(* CoDeSys 2.3.9.47 project: PassiProj_V2_3.pro *)
(* Libraries: Ethernet.lib 2.12.10 14:48:32, SerComm.lib 31.5.11 08:54:36, Serial_Interface_01.lib 22.4.13 12:50:14, SysLibEvent.lib 2.12.10 14:48:34, SysLibFile.lib 2.12.10 14:48:34, SysLibPlcCtrl.lib 2.12.10 14:48:32, SysLibSockets.lib 10.2.11 09:20:54, SysLibRtc.lib 2.12.10 14:48:32, Util.lib 26.9.14 11:12:46, Visual.lib 2.12.10 14:48:34, WagoLibStatus.lib 2.12.10 14:48:32, Standard.lib 2.12.10 14:48:34, SYSLIBCALLBACK.LIB 2.12.10 14:48:32 *)

(* PLC configuration (modules and I/O channels)
releLux1 AT %QX2.0 [BOOLOnX_Q] Ch_1 Digital output
releLux2 AT %QX2.1 [BOOLOnX_Q] Ch_2 Digital output
AT %QX2.2 [BOOLOnX_Q] Ch_3 Digital output
AT %QX2.3 [BOOLOnX_Q] Ch_4 Digital output
LUM01 AT %IW0 [WORDOnW_I] Ch_1 Input word
LUM02 AT %IW1 [WORDOnW_I] Ch_2 Input word
LUM03 AT %IW2 [WORDOnW_I] Ch_1 Input word
LUM04 AT %IW3 [WORDOnW_I] Ch_2 Input word
LUM05 AT %IW4 [WORDOnW_I] Ch_1 Input word
LUM06 AT %IW5 [WORDOnW_I] Ch_2 Input word
LUX01 AT %QW0 [WORDOnW_Q] Ch_1 Analog output
LUX02 AT %QW1 [WORDOnW_Q] Ch_2 Analog output
Fieldbus variables [FB_VARS] node 1, in %IB0 out %QB0
Flag variables [FLAG_VARS] node 2, in %IB0 out %QB0
Modbus-Master [MB_MASTER] node 3, in %IB0 out %QB0
*)

(* Global variable list: Global_Constants *)
VAR_GLOBAL CONSTANT

	Plant_NAME			: STRING :='cySN:128 cyVER:1 - ';
	Plant_SN			: DWORD  :=128;	(* S/N Impianto di telecontrollo *)
	Plant_SW_VER		: WORD   :=1;		(* Versione SW installata *)


	(* Colour defines *)
	COLOR_RED			: DWORD	:= 16#2020F0;
	COLOR_YELLOW		: DWORD	:= 16#20F0F0;
	COLOR_GREEN			: DWORD	:= 16#20F020;
	COLOR_LIGHT_GREEN	: DWORD 	:= 16#006000;
	COLOR_GREEN_OFF	 : DWORD	:= 16#108010;

	(* Parameters *)
	Plant_DefaultTAmb	: INT	:=100;		(* [.1°C] Temperatura ambiente di default in caso di rottura sonda *)
	Plant_MaxRunTAmb	: INT   :=210; 		(* [.1°C] Temperatura ambiente massima funzionamento impianto *)
	Plant_AntiFreezeTAmb: INT   :=-40;		(* [.1°C] Antifreeze temperature, start circulators *)
	Plant_VRD_TAlarm	: INT   :=850;(*450;*) 		(* [.1°C] Temperatura di allarme VRD, blocco *)
	Plant_VRD_TMax		: INT   :=800;(*430;*) 		(* [.1°C] Setpoint massimo per uscita VRD *)
	Plant_VRD_TDefault	: INT	:=300;		(* [.1°C] Temperatura di default in caso di errore climatica *)
	Plant_CirOffDelay	: TIME	:=T#30m;	(* (Def.T#15m) Ritardo spegnimento pompe per ricircolo caldaia *)
	Plant_CirOnDelay	: TIME	:=T#15m;
	Plant_MaxWaterLoss	: WORD  :=2;		(* [lt/h] Massima perdita del circuito *)

	(* Filesystem *)
	FilesPath  			: STRING :='S:\';

	(* TCP Logger *)
	Logger_SERVER		: STRING:='';
	Logger_IP				: STRING:= '192.168.100.3';
	Logger_PORT			: WORD  :=80;
	Logger_GETSTART		: STRING:='GET /cygmsrv/passi.ashx?';
	Logger_GETEND		: STRING:='$R$N$R$N';
	Logger_CHECK		: STRING:='True';
	Logger_CRLF			: STRING:='$R$N';
	Logger_DataFile		: STRING:='S:\LOG.DAT';
	Logger_DataFileOld	: STRING:='S:\LOG.BCK';
	Logger_IndexFile	: STRING:='S:\LOG.IDX';
	Logger_ConnRetries	: BYTE:=5;
	Logger_RecoverMsgs	: BYTE:=25;

	(* TCP Remote *)
	Remote_PORT			: WORD  :=10;
	Remote_WELCOME		: STRING:='Connected$R$N';
	Remote_OK			: STRING:='OK$R$N';
	Remote_ERROR		: STRING:='ERROR$R$N';

	(* TCP Sockets *)
	MAX_SEND_TCP_SERVER					 : DWORD:=12000;(*60000*)
	MAX_RECEIVE_TCP_SERVER				 : DWORD:=12000; (*3000;*)
	MAX_RECEIVE_TCP_SERVER_SOCKET	 	 : DWORD:=12000; (* 1500; *)
	MAX_SEND_TCP_CLIENT					 : DWORD:=12000;(*15000*)
	MAX_RECEIVE_TCP_CLIENT				 : DWORD:=12000;
	MAX_RECEIVE_TCP_CLIENT_SOCKET		 : DWORD:=12000;
	MAX_RECEIVE_UDP_SERVER				 : INT  :=1472;
	MAX_RECEIVE_UDP_CLIENT				 : INT  :=1472;
	CONNECT_WATCHDOG_TIME				 : TIME :=t#10s;


	(*  *)
	MAXLUM : BYTE:=2;  (*  6 *)

	(* Lux element *)
	ANALOG		: BOOL:=0;
	DIGITAL			: BOOL:=1;
	MAX_LUXNUM	: WORD := 2;	(* si prevedono al max 100 - 120 lux *)
	LUXM_MAX_ID	: WORD:=250;
	MAX_ARRAY_MSG	: BYTE:=99;

	CRON_MAX	: WORD := 5;



	(* Dim ARRAY retentivi  *)
	MAX_LUX_RETAIN	: BYTE := 250;
	MIN_FOR_DAY: WORD:=1440;
	DOUBLE_MIN_FOR_DAY: WORD:=2880;
	QUARTER_FOR_DAY:WORD:=96;
	DOUBLE_QUARTER_FOR_DAY:WORD:=192;
END_VAR



VAR_GLOBAL
	TestNodoInterogato: BYTE;
	NodoDaInterrogare: BYTE;
	InibiscoModbus: BOOL;
END_VAR

(* Global variable list: Global_Retain *)
VAR_GLOBAL RETAIN PERSISTENT
	Mode_Manual : BOOL := FALSE;
(*
	GRU01_Clima	: typ_Clima;

	VRD01_Clima : typ_Clima;
	VRD02_Clima : typ_Clima;
	VRD03_Clima : typ_Clima;  *)

	Ctl01_Counter	:	DWORD;
	Ctl02_Counter	:	DWORD;
	Ctl03_Counter	:	DWORD;

(* Impostazioni di imipanto *)

	DelayAllarmeTemperaturaNonRaggiunta: INT;
	DeltaInterventoAllarmeTempeaturaNonRaggiuta: INT;
	OffsetSetPointManuale:INT;							(* Offset al Setpoint manuale per comensare lo scambiatore *)

	SogliaMinStartAntigelo: INT;
	SogliaMinStopAntigelo: INT;
	BitAbilitaAntigelo: BOOL:=TRUE;


	GlobalWorkingtime		: ARRAY [1..MAX_LUX_RETAIN] OF DWORD; (* [sec] Internal working time counter *)
	GlobalPowerOnCycles	: ARRAY [1..MAX_LUX_RETAIN] OF WORD;	(*/DWORD;  *) (* Internal counter of power-on cycles *)
	GlobalEnergyCounter	: ARRAY [1..MAX_LUX_RETAIN] OF WORD; (* DWORD;  *) (* [E-1 kWh] Internal energy counter *)
	GlobalEnergyCounter_t 	: ARRAY [1..MAX_LUX_RETAIN] OF DWORD; (* Temporary energy in E-2*Wsec *)

END_VAR

(* Global variable list: Global_Variables *)
VAR_GLOBAL

	SYS    : typ_SYS;
	Logger : typ_Logger;

	T_AMB	:	INT;		(* Environment temperature *)

	Rampa_1, Rampa_2	: RAMP_INT;
	RampUp			:INT:=500;
	RampDown			:INT:=500;
	RampTime			:TIME:= t#500ms;



	(**** PLANT OBJECTS ****)
	(*...*)
(*	GRU01	:	obj_CAL_VT300GW2 := (ID:=1); *)

	(* Water counter - 2 PULSES/LITER *)

	(* Heat counter *)

	(* Cronothermostat *)
(*	THER01	:	obj_CRONTER := (ID:=1, Local_MaxRunTAmb:=250,Histeresys:=10);
	THER02	:	obj_CRONTER := (ID:=2, Local_MaxRunTAmb:=250,Histeresys:=10);
	THER03	:	obj_CRONTER := (ID:=3, Local_MaxRunTAmb:=250,Histeresys:=10);
	THER04	:	obj_CRONTER := (ID:=4, Local_MaxRunTAmb:=600,Histeresys:=10);	(* There is no an environment probe	*)
	THER05	:	obj_CRONTER := (ID:=5, Local_MaxRunTAmb:=800,Histeresys:=50);	(*  crono per la gestione della caldaia a muro ex CAL04 ora CIR250 *)
	THER250	:	obj_CRONTER := (ID:=250, Local_MaxRunTAmb:=800,Histeresys:=50);	(*  crono per la gestione della caldaia a muro ex CAL04 ora CIR250 *)


	 Boiler *)

	(* Pump *)

	(* Modbus double pumps *)

	(* ModBus Pumps *)

	(* Valves
	VRD01	:	obj_VRD_new 	:= (ID:=1, fFeedback:=TRUE, ReducedRange := TRUE,Local_VRD_TAlarm:=450);
	VRD02	:	obj_VRD_new 	:= (ID:=2, fFeedback:=TRUE, ReducedRange := TRUE,Local_VRD_TAlarm:=450);
	VRD03	:	obj_VRD_new 	:= (ID:=3, fFeedback:=TRUE, ReducedRange := TRUE,Local_VRD_TAlarm:=850);
 *)

	TolleranceLowLux	:WORD :=2; (* Tolleranza per isteresi in Lux - era 25 *)
	TolleranceHighLux	:WORD :=2; (* Tolleranza per isteresi in Lux  - era 25 *)

	(* Lux probes *)
	LumList : ARRAY [1..6] OF obj_LUM;

	LuxElement		: ARRAY [1..MAX_LUXNUM] OF obj_LUX;  (* Lista di variabili Lux   *)

	DataLuxForVis	: ARRAY [1..MAX_LUXNUM] OF type_DataLuxForVis;	(*ARRAY ordinato contenente i valori Status_Vis e del timer utilizzati per la visualizzazione (PLC_Visualization)*)

	LuxOutput		: ARRAY [1..LUXM_MAX_ID] OF type_LuxOutput;

	(* Crono *)
	CRON   			: ARRAY [1..CRON_MAX] OF obj_CRON;
	CronEd			: obj_CRON_EDITOR;
	LuxSuBit		: REAL:= 0.15259;  (* 60000 / 32767= 1.83111 *) (* 5000 / 32767= 0.15259 *)  (* 1000 / 32767= 0.03 *)

	(** Communication **)
	(**** SIMULATION ONLY ****)
	(*...*)END_VAR

(* Data type in Lux *)
TYPE en_ActionKey :
(
	NormalMode 	:= 0,
	SwitchON		:= 1,
	SwitchOFF		:= 2,
	Restore			:= 3
);
END_TYPE

(* Data type in Lux *)
TYPE en_KeyMode :
(
	BUTTON_NO		:=01,
	BUTTON_NC		:=02,
	SWITCH_NO		:=03,
	SWITCH_NC			:=04
);
END_TYPE

(* Data type in Logger *)
TYPE en_Logger_ErrLev :
(
	EL_Log			:=0,
	EL_Wrn			:=1,
	EL_Alarm		:=2,
	EL_AlarmStop	:=3
);
END_TYPE

(* Data type in Logger *)
TYPE en_Logger_Status :
(
	S_Logger_UNKNOWN := 0,
	S_Logger_IDLE,
	S_Logger_WAITCONN,
	S_Logger_WAITTX,
	S_Logger_WAITRESP,
	S_Logger_ERROR
);
END_TYPE

(* Data type in Lux *)
TYPE en_Modality :
(
	ManualeOff 	:= 0,
	ManualeOn 	:= 1,
	Cronografo	:= 2,
	Timer		:= 3,
	KeyControl	:= 4
);
END_TYPE

(* Data type *)
TYPE en_SYS_Objects :
(
	EO_SYS		:=0,  (* PLC *)
	EO_VPN		:=1,  (* VPN *)
	EO_DOOR		:=2,  (* Door & access control *)

	EO_CAL		:=10, (* Caldaia *)
	EO_CIR		:=11, (* Circolatore *)
	EO_CRON		:=12, (* Crono-termostato *)
	EO_VRD		:=13, (* Valvola miscelatore pannelli *)
	EO_CTL		:=14, (* Contalitri *)
	EO_CTB		:=15, (* Contabilizzatore *)
	 (*EO_TPV		:=16, Temperature probes values *)
	EO_PPV		:=17, (* Pressure probes values *)
	EO_PBV		:=18, (* Over-Pressure Alarms *)
	EO_TBV		:=19, (* Over-Temperature Alarms *)
	EO_PMV		:=20, (* Under-Pressure Alarms *)
	EO_GRU		:=21, (* Gruppo termico *)
	EO_PDC		:=22, (* Pompa di calore *)
	EO_SOL		:=23, (* Pannello solare termico *)
	EO_ESOL		:=24, (* Pannello solare fotovoltaico *)
	EO_GAS		:=25, (* Contatore GAS *)
	EO_PORT		:=26, (* Misuratore di portata *)
	EO_FPV		:=27, (* Flow probes values *)
	EO_ANZ		:=28, (* Analizzatore di rete *)
	EO_SCA		:=29, (* Signal Control Alarms *)
	EO_LUX		:=30, (* Base Illumination point *)
	EO_LUXM		:=31, (* Metered Illumination point *)
	EO_PSG		:=32, (* Sensore di passaggio *)
	EO_HVAC		:=33, (* Heating, Ventilating and Air Conditioning *)
	EO_HYGRV	:=34, (* Relative Humidity sensors value *)
	EO_COOV		:=35, (* Carbon Dioxide CO2 sensors value *)
	EO_INV		:=36, (* Inverter *)
	EO_STR		:=37, (* Smart string box *)

	EO_CIRD		:=39, (* Double CIR *)
	EO_ACS		:=40, (* Hot domestic water *)
	EO_FRG		:=41, (* Frigo *)
	EO_THER		:=42, (* Thermostat *)
	EO_CIRM		:=43, (* Modbus CIR *)

	EO_LUM		:=16, (* Lumen *)

	EO_ZGW			:=200,  (* ZigBee - Gateway *)
	EO_ZRM			:=201,	(* ZigBee - Repeater *)
	EO_ZREL			:=202,	(* ZigBee - Actuator rele *)
	EO_ZTHL			:=203,	(* ZigBee - Temperature Sensor *)

	EO_ASGW			:=250,	(* ASi - Gateway *)
	EO_ASCBI		:=251,	(* ASi - Input Board, Ciabatta *)

	EO_LON			:=1000, (* Bus - LON *)
	EO_MODBUS		:=1001, (* Bus - MODBUS *)
	EO_MBUS			:=1002, (* Bus - M-BUS *)
	EO_MODBUS_TCP	:=1003, (* Bus - MODBUS TCP *)

	EO_GENERIC		:=9000, (* Generic dataset *)
	EO_EXPO			:=9001 (* EXPO dataset *)
);
END_TYPE

(* Data type *)
TYPE en_SYS_Status :
(
	S_UNKNOWN  := 0,
	S_STARTUP,
	S_INIT_RTC,
	S_INIT_VAR,
	S_AUTOTEST,
	S_RUNNING,
	S_SHUTDOWN,
	S_HALT
);
END_TYPE

(* Data type in Plant_Objects *)
TYPE typ_Cron_Calendar :
STRUCT
	Profile		: ARRAY[0..384] OF BYTE;
END_STRUCT
END_TYPE

(* Data type in Plant_Objects *)
TYPE typ_Cron_Jolly :
STRUCT
	Start		: DT;
	End			: DT;
	Temp		: WORD;
	Flags		: WORD; (* B0:Enabled B1..B15:Unused *)
END_STRUCT
END_TYPE

(* Data type in Plant_Objects *)
TYPE typ_Cron_Profile :
STRUCT
	Flags		: WORD;
	Setpoint	: ARRAY [0..1439] OF WORD;	(*	Setpoint	: ARRAY [0..95] OF WORD;  *)
END_STRUCT
END_TYPE

(* Data type in Logger *)
TYPE typ_Logger :
STRUCT
	Status		: en_Logger_Status;

	SendReq		: BOOL;
	SendIdx		: DWORD;
	SendData	: ARRAY [0..MAX_SEND_TCP_CLIENT] OF BYTE;
	SendLen		: DINT;

	TData		: ARRAY [0..MAX_SEND_TCP_CLIENT] OF BYTE;
	TLen		: DINT;

	LastIdxPos	: DWORD;

	(* Temporary variables used by objects *)
	s1			: STRING(256);
	i1			: WORD;

END_STRUCT
END_TYPE

(* Data type *)
TYPE typ_SYS :
STRUCT
	Status			: en_SYS_Status;
	Warning			: BOOL;
	Alarm			: BOOL;
	AlarmStop		: BOOL;

	Time_LogString	: STRING;
	Time_Year		: WORD;
	Time_Month		: BYTE;
	Time_Day		: BYTE;
	Time_Hour		: BYTE;
	Time_Minute		: BYTE;
	Time_Min		: BYTE;

	Time_CT_DT		: DT;
	Time_CT_Day		: WORD;
	Time_CT_Quarter	: BYTE;
	Time_CT_Minute		: WORD;

	LastLogs_Idx	: BYTE;
	LastLogs_Dat	: ARRAY[0..5] OF STRING;
	LastLogs_Msg	: ARRAY[0..5] OF STRING;

END_STRUCT
END_TYPE

(* Data type in Lux *)
(* La seguente struttura ha la funzione di collegare l'id del lux con i relativi dati qui indicati *)
(* In tal modo la visualizzazione dello stato dei lux viene eseguita associando l'ID dell'array contenente questa struttura*)

TYPE type_DataLuxForVis :
STRUCT
	VisStatus	: DWORD; (* valori di status_vis   *)
	VisTimer	: TIME;	(* Valori dei timer  *)
	VisMod		: en_Modality; (* Impostazione mode  *)
END_STRUCT
END_TYPE

(* Data type in Lux *)
TYPE type_LuxOutput :
STRUCT
	DigitalOut	:	BOOL;
	AnalogOut	:	WORD;
	TypeOut	:	BOOL;
END_STRUCT
END_TYPE

(* POU PLC_PRG, ST *)
PROGRAM PLC_PRG
VAR
	Timer1: TON; (* Fast controls tick *)
	Timer2: TON; (* Plant control tick *)
	Timer3: TON; (* Logger timer *)
	Timer4: TON; (* Media timer *)

	LumValue			: ARRAY [1..6] OF WORD;
	LumValueSum		: DWORD;
	LumValueMax, LumValueMin	: WORD;
	LumValueAverage	: DWORD;
	LumValueAverageLux	:DWORD;
	LuxDeltaBit, LuxEndBit	:WORD;
	x					: BYTE;
	counter				: WORD;
	LuxCount			: WORD;
	LuxEnInfo	: BOOL;
	ValInCrono	: INT; (* Valore del setpoint del crono *)

	TolleranceLowBit		: WORD;
	TolleranceHighBit		: WORD;
	AnalogOutputBit			:WORD;

	ValInCronoVisu			:ARRAY [1..MAX_LUXNUM] OF INT;
	ValInCronoFromVisu		:ARRAY  [1..MAX_LUXNUM] OF BOOL;
	Temp	:INT;
	LuxStateON: BOOL;
END_VAR
(******************************************************************************
 ****                           MAIN TASK CODE                             ****
 ******************************************************************************

	Network setup:
		IP  = 192.168.100.2 | MSK = 255.255.255.0
		GW	= 192.168.100.1 | DNS = 192.168.100.1
		SNTP = 193.204.114.232 (3600s) ==> 192.168.100.3

*)

(*==============================*)
(*===== Main status machine ====*)
(*==============================*)
MainCtrl();
(*
IF SYS.Status>S_INIT_VAR THEN
	Execute cycle processes
END_IF
 *)
(*==============================*)
(*== System cycle operations ===*)
(*==============================*)
(* Execute TCP processes *)
Logger_Proc();
Remote_Proc();
(* Execute Cron Editor commands *)
CronEd();
END_PROGRAM
ACTION MainCtrl:
CASE Sys.Status OF

	S_STARTUP:
		Sys.Status:=S_INIT_RTC;
		FOR counter := 1 TO MAX_LUXNUM DO
			CRON[counter].ID:=counter;
			LuxElement[counter].ID:=counter;
			LuxElement[counter].CTRL_MODE := 2 ; (* TabDefaultLux[counter].Mode; //copio il mode nella tabella delle variabili dei lux 	*)
			LuxElement[counter].CTRL_MODE_backUp := 2;  (* TabDefaultLux[counter].Mode; //salvo il mode di backup per il ripristina modo	*)
			LuxElement[counter].DimmingType:=1; (* settato a dimming *)
		END_FOR
		FOR x:= 1 TO MAXLUM DO
			LumList[x].ID:= x;
		END_FOR
	S_INIT_RTC:
		(* Check RTC and update from network *)
		RTC_Update();
		(* Check time *)
		IF Sys.Time_Year>2000 THEN
			Sys.Status:=S_INIT_VAR;
		END_IF

	S_INIT_VAR:
		LogEv(EL_Wrn,EO_SYS,0,1,CONCAT('System_startup_v',WORD_TO_STRING(Plant_SW_VER)));
		Sys.Status:=S_RUNNING;

	S_RUNNING:
		Timer1(IN:=NOT Timer1.Q,PT:=T#50ms);
		IF Timer1.Q THEN
			(* Update meters *)

			(* Update system checks *)
			SYS_Proc();
		END_IF

		Timer2(IN:=NOT Timer2.Q,PT:=T#500ms);
		IF Timer2.Q THEN
			(* Read current date/time *)
			RTC_Update();


			(*Lum Probes *)
			IF ValInCronoFromVisu[1] = TRUE THEN
				LumList[1](IN:=LUM01, IN_TARGET:=ValInCronoVisu[1]*10);
			ELSE
				CRON[1]( SetPoint=>ValInCrono);
				LumList[1](IN:=LUM01, IN_TARGET:=ValInCrono);
			END_IF
			IF ValInCronoFromVisu[2] = TRUE THEN
				LumList[2](IN:=LUM02, IN_TARGET:=ValInCronoVisu[2]*10);
			ELSE
				CRON[2]( SetPoint=>ValInCrono);
				LumList[2](IN:=LUM02, IN_TARGET:=ValInCrono);
			END_IF
			LumValue[1]:=LumList[1].AVG;
			LumValue[2]:=LumList[2].AVG;
		(*	LumList[3](IN:=LUM03);
			LumValue[3]:=LumList[3].AVG;
			LumList[4](IN:=LUM04);
			LumValue[4]:=LumList[4].AVG;
			LumList[5](IN:=LUM05);
			LumValue[5]:=LumList[5].AVG;
			LumList[6](IN:=LUM06);
			LumValue[6]:=LumList[6].AVG;
		 *)
			Timer4(IN:=NOT Timer4.Q,PT:=T#500ms);
			IF Timer4.Q THEN
				LumValueSum:=0;
				FOR x:= 1 TO MAXLUM DO
					LumValueSum:= LumValueSum+ LumValue[x];
				END_FOR
				LumValueAverage:=(LumValueSum / MAXLUM);
				LumValueAverageLux:=REAL_TO_DWORD(LumValueAverage*LuxSuBit);
			END_IF

			TolleranceLowBit := REAL_TO_WORD (TolleranceLowLux / LuxSuBit);
			TolleranceHighBit := REAL_TO_WORD (TolleranceHighLux / LuxSuBit);

		FOR LuxCount:=1 TO  MAX_LUXNUM DO
			IF  LuxElement[LuxCount].ID <> 0  THEN (* esegue scansione dei lux dell'impianto solo se presenti *)
	
				CASE LuxElement[LuxCount].CTRL_MODE OF
					0: (* Manuale Off *)
					LuxElement[LuxCount](LuxTypeOut => LuxOutput[LuxCount].TypeOut,
											LuxDigitalOut => LuxOutput[LuxCount].DigitalOut,
											LuxAnalogOut => LuxOutput[LuxCount].AnalogOut,
											Lux_Enable=>LuxEnInfo,
											LocalWorkingTime:=GlobalWorkingtime[LuxCount],
											LocalPowerOnCycles:=GlobalPowerOnCycles[LuxCount],
											LocalEnergyCounter:=GlobalEnergyCounter[LuxCount],
											LocalEnergyCounter_t:=GlobalEnergyCounter_t[LuxCount],KeyQty:=2);
					1:  (* Manuale On *)
					LuxElement[LuxCount](LuxTypeOut => LuxOutput[LuxCount].TypeOut,
											LuxDigitalOut => LuxOutput[LuxCount].DigitalOut,
											LuxAnalogOut => LuxOutput[LuxCount].AnalogOut,
											Lux_Enable=>LuxEnInfo,
											LocalWorkingTime:=GlobalWorkingtime[LuxCount],
											LocalPowerOnCycles:=GlobalPowerOnCycles[LuxCount],
											LocalEnergyCounter:=GlobalEnergyCounter[LuxCount],
											LocalEnergyCounter_t:=GlobalEnergyCounter_t[LuxCount],KeyQty:=2);
					2:	(* se il mode è settato come cronografo gestisco accensione a orologio *)
					CRON[LuxCount]( SetPoint=>ValInCrono);
					(*	LuxElement[LuxCount].ValInCronoInLux:=ValInCrono;   *)
					IF ValInCronoFromVisu[LuxCount] = TRUE THEN
						LuxElement[LuxCount].ValInCronoInLux:=ValInCronoVisu[LuxCount]*10;
					ELSE
						LuxElement[LuxCount].ValInCronoInLux:=ValInCrono;
					END_IF
			(*		KeyTest((*KeyMode:= 01,*)CtrlKey:=LUX_ST[108],Cmd_Enable=>LuxEnInfo );
					KeyTest1((*KeyMode:= 01,*)CtrlKey:=LUX_ST[107],Cmd_Enable=>LuxEnInfo1 );				
					LuxElement[LuxCount].CtrlKeyList[0]:=LuxEnInfo;
					LuxElement[LuxCount].CtrlKeyList[1]:=LuxEnInfo1;								 *)
					LuxElement[LuxCount](LuxTypeOut => LuxOutput[LuxCount].TypeOut,
											LuxDigitalOut => LuxOutput[LuxCount].DigitalOut,
											LuxAnalogOut => LuxOutput[LuxCount].AnalogOut,
											Lux_Enable=>LuxEnInfo,
											LocalWorkingTime:=GlobalWorkingtime[LuxCount],
											LocalPowerOnCycles:=GlobalPowerOnCycles[LuxCount],
											LocalEnergyCounter:=GlobalEnergyCounter[LuxCount],
											LocalEnergyCounter_t:=GlobalEnergyCounter_t[LuxCount],KeyQty:=2);  (*, KeyMode:=KeyTest.KeyMode); *)
				END_CASE
				AnalogOutputBit:= REAL_TO_WORD( LuxOutput[LuxCount].AnalogOut*3.27);
				(* codice non in uso - start *)
				IF  AnalogOutputBit < 3100  THEN
					LuxStateON:=FALSE;	(* se devo aprire il relè per spegnere *)
				ELSIF  AnalogOutputBit  > 3600 THEN
					LuxStateON:=TRUE;	(* se devo chiudere il relè per accendere *)
				END_IF
				(* codice non in uso - end *)
				IF ( AnalogOutputBit > TolleranceLowBit) AND  (AnalogOutputBit < (32767-TolleranceHighBit) ) THEN
					IF  ( LuxOutput[LuxCount].AnalogOut>0 AND
						( ( LumValueAverage<AnalogOutputBit - TolleranceLowBit) OR ( LumValueAverage>AnalogOutputBit + TolleranceHighBit) ))THEN
							IF ( LumValueAverage>AnalogOutputBit + TolleranceHighBit) THEN  (* se il valore medio misurato è maggiore del target impostato  *)
								LuxDeltaBit:=  DWORD_TO_WORD(LumValueAverage)-AnalogOutputBit; (* calcolo diff tra misura e target  *)
								IF LuxDeltaBit < AnalogOutputBit THEN  (* se il delta è minore del target posso sottrarla al target altrimenti azzero l'uscita (posta a 1 bit)  *)
									LuxEndBit:= AnalogOutputBit - LuxDeltaBit;
										(*LuxStateON:=TRUE; se devo chiudere il relè per accendere *)
								ELSE
									 LuxEndBit := 1;
									 (* LuxStateON:=FALSE;	se devo aprire il relè per spegnere *)
								END_IF
								(* LuxEndBit:=REAL_TO_INT(LuxOutput[LuxCount].AnalogOut*3.27) - LuxDeltaBit;  *)
							ELSIF ( LumValueAverage<AnalogOutputBit - TolleranceHighBit) THEN
								LuxDeltaBit:= DWORD_TO_WORD( AnalogOutputBit - LumValueAverage);
								LuxEndBit:= AnalogOutputBit + LuxDeltaBit;
								(* LuxStateON:=TRUE;	 se devo chiudere il relè per accendere *)
								(* LuxEndBit:=REAL_TO_INT(LuxOutput[LuxCount].AnalogOut*3.27) + LuxDeltaBit;  *)
							END_IF;
							CASE LuxCount OF
								1:	IF luxEndBit >32727 THEN
										LuxEndBit:=32727;
									END_IF
									 (*releLux1:=LuxStateON;   apro il contatto del relè se il lux è spento *)
								 	Rampa_1(in:= LuxEndBit, ascend:=RampUp, descend:=RampDown, timebase:=RampTime);
								(*Rampa_1(in:= REAL_TO_INT(LuxOutput[LuxCount].AnalogOut*3.27), ascend:=RampUp, descend:=RampDown, timebase:=RampTime);*)
									 LUX01:=Rampa_1.OUT;

								(*		1: LUX01:= REAL_TO_WORD(LuxOutput[LuxCount].AnalogOut*3.27);	*)
								2:  IF luxEndBit >32727 THEN
										LuxEndBit:=32727;
									END_IF
									 (*releLux1:=LuxStateON;   apro il contatto del relè se il lux è spento *)
									Rampa_2(in:= LuxEndBit, ascend:=RampUp, descend:=RampDown, timebase:=RampTime);
								(*Rampa_2(in:= REAL_TO_INT(LuxOutput[LuxCount].AnalogOut*3.27), ascend:=RampUp, descend:=RampDown, timebase:=RampTime);*)
									 LUX02:=Rampa_2.OUT;
								(*		 LUX02:= REAL_TO_WORD(LuxOutput[LuxCount].AnalogOut*3.27);	*)
							END_CASE;

					END_IF
				ELSIF ( (AnalogOutputBit > (32767-TolleranceHighBit) ) OR ( AnalogOutputBit < TolleranceLowBit) ) THEN
						CASE LuxCount OF
							1: Rampa_1(in:= REAL_TO_INT(LuxOutput[LuxCount].AnalogOut*3.27), ascend:=RampUp, descend:=RampDown, timebase:=RampTime);
								 LUX01:=Rampa_1.OUT;
							2: Rampa_2(in:= REAL_TO_INT(LuxOutput[LuxCount].AnalogOut*3.27), ascend:=RampUp, descend:=RampDown, timebase:=RampTime);
								 LUX02:=Rampa_2.OUT;
						END_CASE;
				END_IF
(*
				IF Rampa_1.OUT  < 3000  OR Rampa_2.OUT < 3000 THEN (* 3100 *)
					releLux1:=FALSE;
				ELSIF( Rampa_1.OUT >3200 OR Rampa_2.OUT > 3200) THEN  (*  3600 *)
					 releLux1:=TRUE;
				END_IF
 *)
				IF (Rampa_1.OUT  < 3000)  THEN (* 3100 *)
					releLux1:=FALSE;
				ELSIF( Rampa_1.OUT >3200 ) THEN  (*  3600 *)
					 releLux1:=TRUE;
				END_IF
				IF (Rampa_2.OUT  < 3000)  THEN (* 3100 *)
					releLux2:=FALSE;
				ELSIF( Rampa_2.OUT >3200 ) THEN  (*  3600 *)
					 releLux2:=TRUE;
				END_IF

			END_IF
		END_FOR



			(* Test toggle *)
			(*IF TEST1 THEN TEST1:=FALSE; ELSE TEST1:=TRUE; END_IF*)
		END_IF

		Timer3(IN:=NOT Timer3.Q,PT:=T#1m);
		IF Timer3.Q THEN
			(* Trig logger *)
			LogTrig();
			(* Execute temporary CSV logger *)
			(*CSV_Log();*)
		END_IF

	S_SHUTDOWN:
		(* Stop sistema *)
		Sys.Status:=S_STARTUP;

	S_HALT:
		(* Aspetta uscita manuale *)
		Sys.Status:=S_STARTUP;

	S_UNKNOWN:
	Sys.Status:=S_STARTUP;
ELSE
	Sys.Status:=S_STARTUP;
END_CASE;
END_ACTION

(* POU TCP_Logger/Logger_Proc, ST *)
PROGRAM Logger_Proc
VAR
	c1:         	TCPCLIENT;

	Open:	    	BOOL;
	IpAddr:			DWORD;
	InetAddr:		DWORD;
	Connected:  	BOOL;
	Error:      	DINT;
	TxTrig:     	BOOL;
	RxData:			ARRAY [0..MAX_RECEIVE_TCP_CLIENT] OF BYTE;
	RxLen:			DINT;

	Retry:			BYTE;	(* Counter for connection retries *)
	Recovered:		BYTE;	(* Counter for recovered unsent messages *)

	i:				DINT;
	pos:			DWORD;
	hFile:			DWORD;

END_VAR
(*=== State machine ===*)
CASE Logger.Status OF

	S_Logger_UNKNOWN:
		(* Startup *)
		Logger.SendReq:=FALSE;
		Open:=FALSE;
		Logger.Status:=S_Logger_IDLE;

	S_Logger_IDLE:
		(* Wait request *)
		IF Logger.SendReq THEN
			(* Resolve server name or use static IP *)
			IF LEN(Logger_SERVER)=0 THEN
				InetAddr:=SysSockInetAddr(Logger_IP);
			ELSE
				IpAddr:=SysSockGetHostByName(ADR(Logger_SERVER));
				DWORDSWAP(pIn:=ADR(IpAddr), pOut:=ADR(InetAddr));
			END_IF
			TxTrig:=FALSE;
			RxLen:=0;
			(* Open connection *)
			Open:=TRUE;
			Logger.Status:=S_Logger_WAITCONN;
		END_IF

	S_Logger_WAITCONN:
		(* Wait connection *)
		IF Connected THEN
			(* Send data *)
			TxTrig:=TRUE;
			Logger.Status:=S_Logger_WAITTX;
		END_IF
		IF Error>0 THEN
			Open:=FALSE;
			Logger.Status:=S_Logger_ERROR;
		END_IF

	S_Logger_WAITTX:
		(* Wait transmission *)
		IF NOT TxTrig THEN
			Logger.Status:=S_Logger_WAITRESP;
		END_IF
		IF Error>0 THEN
			Open:=FALSE;
			Logger.Status:=S_Logger_ERROR;
		END_IF

	S_Logger_WAITRESP:
		(* Wait response *)
		IF Connected=FALSE (* OR TIMEOUT!! *) THEN
			Open:=FALSE;
			(* Check response *)
			IF RxLen>=4 AND CHKSTRING(pString:=ADR(RxData), pPattern:=ADR(Logger_CHECK)) THEN
				Logger.SendReq:=FALSE;
				Retry:=0;
				(* Check unsent messages to flush *)
				IF Recovered<Logger_RecoverMsgs THEN
					MsgChk();
					IF Logger.SendReq=TRUE THEN
						Recovered:=Recovered+1;
					ELSE
						Recovered:=0;
					END_IF
				ELSE
					Recovered:=0;
				END_IF
				Logger.Status:=S_Logger_IDLE;
			ELSE
				Logger.Status:=S_Logger_ERROR;
			END_IF
		END_IF

	S_Logger_ERROR:
		(* Connection error or send failure *)
		Retry:=Retry+1;
		IF Retry>Logger_ConnRetries THEN
			(* Save message as unsent *)
			MsgSave();
			Logger.SendReq:=FALSE;
			Retry:=0;
		END_IF
		Logger.Status:=S_Logger_IDLE;

ELSE
	Logger.Status:=S_Logger_UNKNOWN;
END_CASE


(*=== Execute client lib ===*)
c1(
	xOpenConnection			:= Open,
	dwInetAddr 				:= InetAddr,
	wPortNumber				:= Logger_PORT,
	ptSendData				:= ADR(Logger.SendData),
	diSendCount				:= Logger.SendLen,
	tConnectWatchdogTime	:= t#10s,
	xStartSend				:= TxTrig,
	aReceiveBuffer			:= RxData,
	diReceiveCount			:= RxLen,
	xConnected				=> Connected,
	diError					=> Error
);

(*=== Process Rx data ===*)
(*IF RxLen>0 THEN
	RxLen:=0;
END_IF*)
END_PROGRAM
ACTION MsgChk:
(* Open index file *)
hFile:=SysFileOpen(Logger_IndexFile,'r');
IF hFile=0 THEN
	RETURN;
END_IF
(* Search oldest message to recover *)
SysFileSetPos(hFile,Logger.LastIdxPos);
Logger.SendLen:=0;
REPEAT
	SysFileRead(hFile, ADR(Logger.SendIdx), SIZEOF(Logger.SendIdx));
	pos:=SysFileGetPos(hFile);
	SysFileRead(hFile, ADR(Logger.SendLen), SIZEOF(Logger.SendLen));
UNTIL
	SysFileEOF(hFile) OR Logger.SendLen<>0
END_REPEAT
SysFileClose(hFile);
(* Delete index file when all messages are recovered *)
IF Logger.SendLen=0 THEN
	Logger.LastIdxPos:=0;
	SysFileDelete(Logger_IndexFile);
	RETURN;
END_IF
(* Recover message data *)
hFile:=SysFileOpen(Logger_DataFile,'r');
IF hFile<>0 THEN
	SysFileSetPos(hFile,Logger.SendIdx);
	SysFileRead(hFile,ADR(Logger.SendData),Logger.SendLen);
	Logger.SendReq:=TRUE;
	SysFileClose(hFile);
END_IF
(* Clear index entry *)
hFile:=SysFileOpen(Logger_IndexFile,'a');
IF hFile<>0 THEN
	SysFileSetPos(hFile,pos);
	i:=0;
	SysFileWrite(hFile, ADR(i), 4);
	Logger.LastIdxPos:=SysFileGetPos(hFile);
	SysFileClose(hFile);
END_IF
END_ACTION
ACTION MsgSave:
(* Add log position in recovery indexes *)
hFile:=SysFileOpen(Logger_IndexFile,'a');
SysFileWrite(hFile, ADR(Logger.SendIdx), SIZEOF(Logger.SendIdx));
SysFileWrite(hFile, ADR(Logger.SendLen), SIZEOF(Logger.SendLen));
SysFileClose(hFile);
END_ACTION

(* POU Utils Functions/TCPCLIENT, ST *)
FUNCTION_BLOCK TCPCLIENT
(***********************************************************************************************************	*)
(* Version: 1.3b                        			          													*)
(* Date: 28.10.2014                   				          							            			*)
(***********************************************************************************************************	*)
(* WAGO Kontakttechnik GmbH Hansastr. 27 32423 Minden(Westf.)													*)
(* Tel. +0049 571/887-0 Fax. +0049 571/887-0																	*)
(* Author: VB																									*)
(***********************************************************************************************************	*)
(*Description:	A TCP client to read and write data with additional connection watchdog							*)
(*History:																										*)
(*Version 1.3b: 28.10.2014: Use DWORD address for IP (Andrea Ravasio)											*)
(*Version 1.3: 11.02.2011: Changes according to 750-880/881											 			*)
(*Version 1.2: 29.08.2007 Bugfix TCP Client																		*)
(*Version 1.1: 15.01.2007 Changes according to FW11																*)
(*Version 1.0: 09.03.2006 Release																				*)
(***********************************************************************************************************	*)
VAR CONSTANT
	STATE_CREATE     				 : BYTE:= 0;
	STATE_OPEN     					 : BYTE:= 1;
	STATE_IOCTL    					 : BYTE:= 2;
	STATE_CONNECT     				 : BYTE:= 10;
	STATE_TX       					 : BYTE:= 20;
	STATE_RX       					 : BYTE:= 30;
	STATE_CLOSE    					 : BYTE:= 40;
	STATE_ERROR_TRAP			     : BYTE:= 200;
END_VAR

VAR_INPUT
	xOpenConnection					: BOOL;
	dwInetAddr						: DWORD; (* <== Use SysSockInetAddr() value or
													swapped bytes order of SysSockGetHostByName() value *)
	wPortNumber						: WORD;
	ptSendData						: POINTER TO ARRAY[0..MAX_SEND_TCP_CLIENT] OF BYTE;
	diSendCount						: DINT;
	tConnectWatchdogTime		    : TIME := t#10s;
END_VAR
VAR_OUTPUT
	xConnected						: BOOL;
	diError 						: DINT := 0;
END_VAR
(* ErrorCodes -----------------------------------------
	16#8001 => No socket descriptor available 
	16#8002 => SysSockSend returns -1 
	16#8003 => Socket was "gracefully closed" 
	16#8004 => switching to none blocking mode fails
	16#8005 => SysSockClose() returns FALSE 
    16#8006 => SysSockConnect() fails
    16#8007 => SysSockSend() fails
	16#8008 => error state machine 
	16#8009 => timeout while waiting for data from server 
------------------------------------------------------------*)
VAR_IN_OUT
	xStartSend							: BOOL;
	aReceiveBuffer						: ARRAY [0..MAX_RECEIVE_TCP_CLIENT] OF BYTE;
	diReceiveCount						: DINT;
END_VAR
VAR
	m_State								: BYTE := 0;
	m_ReceiveBuffer						: ARRAY [0..MAX_RECEIVE_TCP_CLIENT_SOCKET] OF BYTE;
	m_Socket							: DINT;
	m_AddressInfo						: SOCKADDRESS;
	m_BytesReceived						: DINT;
	m_diReturn							: DINT;
	m_xReturn							: BOOL;
	m_IoCtlParameter  					: DINT := 1; (* IOCTL-Parameter for non-blocking mode of sockets *)
	i									: INT;
	T_Connect							: TON;
	m_count								: DINT;
	diOption							: DINT := 1;
	m_Blocking   						: DINT := 0;
END_VAR
IF xOpenConnection THEN
	(* State maschine *)
	CASE  m_State OF

	(* -------------------------------------------------------------------------*)
	STATE_CREATE:
			(* create socket descriptor*)
			m_Socket := SysSockCreate(diAddressFamily	:= SOCKET_AF_INET,
													 diType		:= SOCKET_STREAM,
													 diProtocol := SOCKET_IPPROTO_TCP);
			IF m_Socket >= 0 THEN
			(*Set Push-Bit*)
				IF ADR(%MW0)=16#30000000  OR ADR(%MW0)=16#20000000 THEN (*841 or 881*)
					SysSockSetOption(
						diSocket:=m_Socket,
						diLevel:=6,
						diOption:=SOCKET_TCP_NODELAY,
						pOptionValue:=ADR(diOption),
						diOptionLength:=SIZEOF(diOption));
				ELSE
						;
				END_IF
				m_State := STATE_IOCTL; (* succesful *)
			ELSE
				diError := 16#8001;  (* no socket descriptor available *)
				m_State := STATE_ERROR_TRAP;
			END_IF

	(* -------------------------------------------------------------------------*)
	STATE_IOCTL: (* change  socket mode  to none blocking *)
		m_diReturn := SysSockIoctl( m_Socket, SOCKET_FIONBIO, ADR(m_IoCtlParameter));
		IF m_diReturn <> 0 THEN
			m_AddressInfo.sin_family := SOCKET_AF_INET;
			m_AddressInfo.sin_port := SysSockNtohs(wPortNumber);
			m_AddressInfo.sin_addr := dwInetAddr;
			m_State := STATE_CONNECT;
		ELSE
			diError := 16#8004;  (* switching to none blocking mode fails *)
			m_State := STATE_ERROR_TRAP;
		END_IF


	(* -------------------------------------------------------------------------*)
	STATE_CONNECT: (* connect with server *)
		T_Connect(IN:=TRUE , PT:=tConnectWatchdogTime);(*activate watchdog for establishing connection to a server*)
		m_xReturn := SysSockConnect ( m_Socket, ADR(m_AddressInfo),  SIZEOF(m_AddressInfo));
		IF m_xReturn THEN (* succesful *)
			IF xStartSend THEN
				m_State := STATE_TX;(*transmit data*)
			ELSE
				m_State := STATE_RX;(*wait for data from server*)
			END_IF
			xConnected:=TRUE;
			T_Connect(IN:=FALSE);
		ELSE
			IF T_Connect.Q THEN
				diError := 16#8006;  (* connect fails *)
				xConnected:=FALSE;
				T_Connect(IN:=FALSE);
				m_State := STATE_ERROR_TRAP;
				SysSockClose( m_Socket);
			ELSE
				m_State := STATE_CONNECT;(*client still  tries to set up connection*)
			END_IF
		END_IF


	STATE_TX:	 (* send TCP-message *)
		m_diReturn := SysSockSend(diSocket := m_Socket,
								  pbyBuffer := ADR(ptSendData^[0]),
								  diBufferSize := diSendCount-m_count,
								  diFlags := 0);

		CASE m_diReturn OF
		-1:	(* ERROR *)
			T_Connect(IN:=TRUE , PT:=CONNECT_WATCHDOG_TIME);(*activate watchdog to check communication*)
			IF t_Connect.Q THEN
				diError := 16#8007;
				T_Connect(IN:=FALSE);
				m_State:=STATE_CLOSE;
			END_IF
		0: (* socket was "gracefully closed" *)
			m_State := STATE_CLOSE;
			diError := 16#8003;
		ELSE (* succesful *)
			m_count:=m_count+m_diReturn;
			IF m_count>=diSendCount THEN
				diError := 16#0000;
				m_State := STATE_RX;
				m_count:=0;
				xStartSend:=FALSE;
			END_IF
			T_Connect(IN:=FALSE);
		END_CASE

	(* -------------------------------------------------------------------------*)
	STATE_RX: (* process receive data *)
			m_BytesReceived := SysSockRecv(	diSocket 	:= m_Socket,
										pbyBuffer 	:= ADR(m_ReceiveBuffer),		(* Address of receive buffer *)
										diBufferSize:= SIZEOF(m_ReceiveBuffer),
										diFlags		:= 0);

			CASE m_BytesReceived OF
			-1:	(* No data available or error occured *)
				T_Connect(IN:=TRUE , PT:=tConnectWatchdogTime);(*activate watchdog to check communication*)
				IF t_Connect.Q THEN
					diError:=16#8009;
					T_Connect(IN:=FALSE);
					m_State:=STATE_CLOSE;
				END_IF
				IF xStartSend THEN
					m_State:=STATE_TX	;(* WAIT IN THIS STATE  and check for arriving data or new send command*)
				END_IF;
			0: (* socket was "gracefully closed"  *)
				m_State:=STATE_CLOSE;
				diError := 16#8003;
			ELSE (* succesful *)
				diError := 16#0000;
				T_Connect(IN:=FALSE);
				(* Copy received data into receive buffer *)
				FOR i:= 0 TO DINT_TO_INT(m_BytesReceived	)-1 DO
					aReceiveBuffer[diReceiveCount]:= m_ReceiveBuffer[i];
					diReceiveCount:=(diReceiveCount+1) MOD SIZEOF(aReceiveBuffer);
				END_FOR

			END_CASE

	(* -------------------------------------------------------------------------*)
	STATE_CLOSE : (* close socket *)
		IF ADR(%MW0)=16#30000000  OR ADR(%MW0)=16#20000000 THEN (*841 or 881*)
			;
		ELSE
			SysSockShutdown(m_Socket, 0);;(*870*)
		END_IF
		m_xReturn := SysSockClose( m_Socket);
		m_Socket := -1;
		m_State := 0; (* succesful *)
		xConnected:=FALSE;
		T_Connect(IN:=FALSE);
	(* -------------------------------------------------------------------------*)
	STATE_ERROR_TRAP: (* error handling *)
		xConnected:=FALSE;

	ELSE  (* Bad FSM code trap  *)
			m_State:= STATE_ERROR_TRAP;
			diError:= 16#8008;
	END_CASE

ELSE(*close connection*)
	IF m_Socket >= 0 THEN
		IF ADR(%MW0)=16#30000000  OR ADR(%MW0)=16#20000000 THEN (*841 or 881*)
			;
		ELSE
			SysSockShutdown(m_Socket, 0);;(*870*)
		END_IF
		SysSockClose( m_Socket);
	END_IF
	m_Socket := -1;
	diError := 16#0000;
	m_State := STATE_CREATE;
	xConnected:=FALSE;
	T_Connect(IN:=FALSE);
END_IF
END_FUNCTION_BLOCK

(* POU Utils Functions/DWORDSWAP, ST *)
FUNCTION DWORDSWAP:BOOL
VAR_INPUT
	pIn:POINTER TO ARRAY[1..4] OF BYTE;
	pOut:POINTER TO ARRAY[1..4] OF BYTE;
END_VAR
VAR
END_VAR
pOut^[1]:=pIn^[4];
pOut^[2]:=pIn^[3];
pOut^[3]:=pIn^[2];
pOut^[4]:=pIn^[1];
END_FUNCTION

(* POU Utils Functions/CHKSTRING, ST *)
FUNCTION CHKSTRING : BOOL
VAR_INPUT
	pString: POINTER TO BYTE;
	pPattern: POINTER TO BYTE;
END_VAR
VAR
END_VAR
CHKSTRING:=TRUE;
WHILE pPattern^<>0 AND CHKSTRING DO
	IF pPattern^<>pString^ THEN CHKSTRING:=FALSE; END_IF
	pString:=pString+1;
	pPattern:=pPattern+1;
END_WHILE
END_FUNCTION

(* POU TCP_Remote/Remote_Proc, ST *)
PROGRAM Remote_Proc
VAR
	s1:         	TCPSERVER;
	Enable: 		BOOL;
	Connected: 		BOOL;
	Error: 			DINT;

	TxData:			ARRAY [0..MAX_SEND_TCP_SERVER] OF BYTE;
	TxLen:			DINT;
	TxTrig:			BOOL;

	RxData:			ARRAY [0..MAX_RECEIVE_TCP_SERVER] OF BYTE;
	RxLen:			DINT;

	Status:			DINT;

	(* Command interpreter *)

	Cmd_Buf:		ARRAY [0..MAX_RECEIVE_TCP_SERVER] OF BYTE;
	Cmd_Buf_U16:	POINTER TO WORD;
	Cmd_Buf_INT:	POINTER TO INT;
	Cmd_BufLen:		WORD;
	Cmd_St:			WORD;

	Cmd_Obj:		WORD;
	Cmd_ObjIdx:		WORD;
	Cmd_C:			WORD;
	Cmd_R:			WORD;
	Cmd_CLen:		WORD;
	Cmd_RLen:		WORD;

	i : WORD;
	j : INT;
	s2 : STRING;


		(* per aggiornare la data e l'ora *)
	SetAnno: INT;
	SetMese: INT;
	SetGiorno: INT;
	SetOra: INT;
	SetMinuti: INT;
	SetSecondi: INT;

		(* per Lux *)
	x	: WORD;
	NewValueTimerH, NewValueTimerL: WORD;
	NewValueTimer: DWORD;
	ModeFromPlc	: WORD;

	temp: WORD;

END_VAR
(*=== State machine ===*)
CASE Status OF
	0: (* Startup *)
		TxLen:=0; TxTrig:=FALSE;
		RxLen:=0;
		Enable:=TRUE;
		Status:=1;

	1: (* Wait incoming connection *)
		IF Connected THEN
			(* Log access *)(*
			LogEv(EL_Log,EO_VPN,1,5,'Remote');*)
			(* Send welcome message *)(*
			ADDSTRING(pTxData:=ADR(TxData), pString:=ADR(Remote_WELCOME), TxLen:=TxLen);
			TxTrig:=TRUE;*)
			(* Reset vars *)
			Cmd_BufLen:=0;
			Cmd_St:=0;
			Status:=2;
		END_IF
		IF Error>1 THEN
			Enable:=FALSE;
			Status:=0;
		END_IF

	2: (* Wait command *)
		IF RxLen>0 THEN
			(*=== Interpreter start ===*)
			IF Cmd_BufLen+(RxLen/2)>=MAX_RECEIVE_TCP_SERVER THEN
				(* ERROR *)
				Cmd_BufLen:=0;
			ELSE
				i:=HEXTORAW(pString:=ADR(RxData), StringLen:=DINT_TO_WORD(RxLen), pData:=ADR(Cmd_Buf[Cmd_BufLen]));
				Cmd_BufLen:=Cmd_BufLen+i;
			END_IF
			IF Cmd_BufLen>=8 THEN
				Cmd_Buf_U16:=ADR(Cmd_Buf[6]);
				IF Cmd_BufLen>=(8+Cmd_Buf_U16^) THEN
					Cmd_CLen:=Cmd_Buf_U16^;
					Cmd_Buf_U16:=ADR(Cmd_Buf[0]); Cmd_Obj:=Cmd_Buf_U16^;
					Cmd_Buf_U16:=ADR(Cmd_Buf[2]); Cmd_ObjIdx:=Cmd_Buf_U16^;
					Cmd_Buf_U16:=ADR(Cmd_Buf[4]); Cmd_C:=Cmd_Buf_U16^;
					(* Log command *)(*
					s2:='RCmd_';		s2:=CONCAT(s2,WORD_TO_STRING(Cmd_Obj));
					s2:=CONCAT(s2,'_'); s2:=CONCAT(s2,WORD_TO_STRING(Cmd_ObjIdx));
					s2:=CONCAT(s2,'_'); s2:=CONCAT(s2,WORD_TO_STRING(Cmd_C));
					s2:=CONCAT(s2,'_');	s2:=CONCAT(s2,WORD_TO_STRING(Cmd_CLen));
					LogEv(EL_Log,EO_VPN,1,6,s2);*)
					(* Execute command *)
					Command();
					Cmd_BufLen:=0;
				END_IF
			END_IF
			(*=== Interpreter end ===*)
			RxLen:=0;
		END_IF
		IF NOT Connected THEN
			Status:=0;
		END_IF

ELSE
	Status:=0;
END_CASE


(*=== Execute server lib ===*)
s1(
	xEnable				:= Enable,
	wPortNumber			:= Remote_PORT,
	tServerTimeOut		:= t#15m,
	ptSendData			:= ADR(TxData),
	diSendCount			:= TxLen,
	xStartSend			:= TxTrig,
	aReceiveBuffer		:= RxData,
	diReceiveCount		:= RxLen,
	xClientConnected	=> Connected,
	diError				=> Error
);
END_PROGRAM
ACTION Cmd_CAL:
(* Check index *)
(*IF Cmd_ObjIdx<>1 THEN
	Cmd_R:=2;
	RETURN;
END_IF

(* Process command *)
CASE Cmd_C OF

	1: (* GET CLIMATIC *)
		Cmd_RLen:=20;
		FOR i:=0 TO 4 DO
			j:=DINT_TO_INT(CAL01_Clima.Points[i].X);
			TxLen:=TxLen+RAWTOHEX(ADR(j),2,ADR(TxData[TxLen]));
			j:=DINT_TO_INT(CAL01_Clima.Points[i].Y);
			TxLen:=TxLen+RAWTOHEX(ADR(j),2,ADR(TxData[TxLen]));
		END_FOR

	2: (* SET CLIMATIC *)
		IF Cmd_CLen<>20 THEN
			Cmd_R:=4;
		ELSE
			FOR i:=0 TO 4 DO
				Cmd_Buf_INT:=ADR(Cmd_Buf[8+4*i]); j:=Cmd_Buf_INT^;
				CAL01_Clima.Points[i].X:=INT_TO_DINT(j);
				Cmd_Buf_INT:=ADR(Cmd_Buf[10+4*i]); j:=Cmd_Buf_INT^;
				CAL01_Clima.Points[i].Y:=INT_TO_DINT(j);
			END_FOR
		END_IF

ELSE
	Cmd_R:=3;
END_CASE*)
;
END_ACTION
ACTION Cmd_CIR:
RETURN;
(*
IF Cmd_ObjIdx<1 OR Cmd_ObjIdx>250 THEN
	Cmd_R:=2;
	RETURN;
END_IF

(* Process command *)
CASE Cmd_C OF

	1:	(* Force CIR On *)
		CASE Cmd_ObjIdx OF

			1:	CIR01.CIR_RUN_REQ := TRUE;
				CIR01.CIR_STOP_REQ 	:= FALSE;
			2:	CIR02.CIR_RUN_REQ := TRUE;
				CIR02.CIR_STOP_REQ 	:= FALSE;
			3:	CIR03.CIR_RUN_REQ := TRUE;
				CIR03.CIR_STOP_REQ 	:= FALSE;
			4:	CIR04.CIR_RUN_REQ := TRUE;
				CIR04.CIR_STOP_REQ 	:= FALSE;
			250:CAL04.CIR_RUN_REQ := TRUE;
				CAL04.CIR_STOP_REQ 	:= FALSE;

		END_CASE

	2:	(* Force CIR Off *)
		CASE Cmd_ObjIdx OF

			1:	CIR01.CIR_STOP_REQ := TRUE;
				CIR01.CIR_RUN_REQ	:= FALSE;
			2:	CIR02.CIR_STOP_REQ := TRUE;
				CIR02.CIR_RUN_REQ	:= FALSE;
			3:	CIR03.CIR_STOP_REQ := TRUE;
				CIR03.CIR_RUN_REQ	:= FALSE;
			4:	CIR04.CIR_STOP_REQ := TRUE;
				CIR04.CIR_RUN_REQ	:= FALSE;
			250:CAL04.CIR_STOP_REQ := TRUE;
				CAL04.CIR_RUN_REQ	:= FALSE;
		END_CASE

	3:	(* Release force *)
		CASE Cmd_ObjIdx OF

			1:	CIR01.CIR_RUN_REQ	:= FALSE;
				CIR01.CIR_STOP_REQ 	:= FALSE;
			2:	CIR02.CIR_RUN_REQ	:= FALSE;
				CIR02.CIR_STOP_REQ 	:= FALSE;
			3:	CIR03.CIR_RUN_REQ	:= FALSE;
				CIR03.CIR_STOP_REQ 	:= FALSE;
			4:	CIR04.CIR_RUN_REQ	:= FALSE;
				CIR04.CIR_STOP_REQ 	:= FALSE;
			250:CAL04.CIR_RUN_REQ	:= FALSE;
				CAL04.CIR_STOP_REQ 	:= FALSE;

		END_CASE

	4: (* SET Tempi delay On Off Circolatori  *)
		CASE Cmd_ObjIdx OF
			1:	Cmd_Buf_U16:=ADR(Cmd_Buf[8]);
				CIR01.OnDelay := DWORD_TO_TIME((Cmd_Buf_U16^)*60*1000); 			(* Delay ON*)
				Cmd_Buf_U16:=ADR(Cmd_Buf[10]);
				CIR01.OffDelay := DWORD_TO_TIME((Cmd_Buf_U16^)*60*1000);			(* Delay OFF *)
			2:	Cmd_Buf_U16:=ADR(Cmd_Buf[8]);
				CIR02.OnDelay := DWORD_TO_TIME((Cmd_Buf_U16^)*60*1000);			(* Delay ON*)
				Cmd_Buf_U16:=ADR(Cmd_Buf[10]);
				CIR02.OffDelay := DWORD_TO_TIME((Cmd_Buf_U16^)*60*1000);			(* Delay OFF *)
			3:	Cmd_Buf_U16:=ADR(Cmd_Buf[8]);
				CIR03.OnDelay := DWORD_TO_TIME((Cmd_Buf_U16^)*60*1000);			(* Delay ON*)
				Cmd_Buf_U16:=ADR(Cmd_Buf[10]);
				CIR03.OffDelay := DWORD_TO_TIME((Cmd_Buf_U16^)*60*1000);			(* Delay OFF *)
			4:	Cmd_Buf_U16:=ADR(Cmd_Buf[8]);
				CIR04.OnDelay := DWORD_TO_TIME((Cmd_Buf_U16^)*60*1000);			(* Delay ON*)
				Cmd_Buf_U16:=ADR(Cmd_Buf[10]);
				CIR04.OffDelay := DWORD_TO_TIME((Cmd_Buf_U16^)*60*1000);			(* Delay OFF *)
		END_CASE


	5: (* GET Tempi delay On Off Circolatori *)
		Cmd_RLen:=4;
			CASE Cmd_ObjIdx OF

			1:	j:=DWORD_TO_WORD(TIME_TO_DWORD((CIR01.OnDelay)/60/1000));
				TxLen:=TxLen+RAWTOHEX(ADR(j),2,ADR(TxData[TxLen]));
				j:=DWORD_TO_WORD(TIME_TO_DWORD((CIR01.OffDelay)/60/1000));
				TxLen:=TxLen+RAWTOHEX(ADR(j),2,ADR(TxData[TxLen]));
			2: 	j:=DWORD_TO_WORD(TIME_TO_DWORD((CIR02.OnDelay)/60/1000));
				TxLen:=TxLen+RAWTOHEX(ADR(j),2,ADR(TxData[TxLen]));
				j:=DWORD_TO_WORD(TIME_TO_DWORD((CIR02.OffDelay)/60/1000));
				TxLen:=TxLen+RAWTOHEX(ADR(j),2,ADR(TxData[TxLen]));
			3: 	j:=DWORD_TO_WORD(TIME_TO_DWORD((CIR03.OnDelay)/60/1000));
				TxLen:=TxLen+RAWTOHEX(ADR(j),2,ADR(TxData[TxLen]));
				j:=DWORD_TO_WORD(TIME_TO_DWORD((CIR03.OffDelay)/60/1000));
				TxLen:=TxLen+RAWTOHEX(ADR(j),2,ADR(TxData[TxLen]));
			4: 	j:=DWORD_TO_WORD(TIME_TO_DWORD((CIR04.OnDelay)/60/1000));
				TxLen:=TxLen+RAWTOHEX(ADR(j),2,ADR(TxData[TxLen]));
				j:=DWORD_TO_WORD(TIME_TO_DWORD((CIR04.OffDelay)/60/1000));
				TxLen:=TxLen+RAWTOHEX(ADR(j),2,ADR(TxData[TxLen]));
		END_CASE


	6: (* LEGGO ALLARME PRESENTE SUL CIRCOLATORE *)
		Cmd_RLen:=2;
			CASE Cmd_ObjIdx OF
			2:	j:=(CIR02.DataPump.PumpAlarm[0]);
				TxLen:=TxLen+RAWTOHEX(ADR(j),2,ADR(TxData[TxLen]));
			3:	j:=(CIR03.DataPump.PumpAlarm[0]);
				TxLen:=TxLen+RAWTOHEX(ADR(j),2,ADR(TxData[TxLen]));

		END_CASE







ELSE
	Cmd_R:=3;
END_CASE
*)
END_ACTION
ACTION Cmd_CIRD:
RETURN;
(*
IF Cmd_ObjIdx<>1 THEN
	Cmd_R:=2;
	RETURN;
END_IF

(* Process command *)
CASE Cmd_C OF

	1:	(* Force CIR On *)
		CIRD01.CIR_RUN_REQ := TRUE;

	2:	(* Force CIR Off *)
		CIRD01.CIR_STOP_REQ := TRUE;

	3:	(* Release force *)
		CIRD01.CIR_RUN_REQ	:= FALSE;
		CIRD01.CIR_STOP_REQ := FALSE;

	4: (* SET Tempi delay On Off Circolatori  *)
		CASE Cmd_ObjIdx OF
			1:	Cmd_Buf_U16:=ADR(Cmd_Buf[8]);
				CIRD01.OnDelay := DWORD_TO_TIME((Cmd_Buf_U16^)*60*1000); 			(* Delay ON*)
				Cmd_Buf_U16:=ADR(Cmd_Buf[10]);
				CIRD01.OffDelay := DWORD_TO_TIME((Cmd_Buf_U16^)*60*1000);			(* Delay OFF *)
		END_CASE


	5: (* GET Tempi delay On Off Circolatori *)
		Cmd_RLen:=4;
			CASE Cmd_ObjIdx OF

			1:	j:=DWORD_TO_WORD(TIME_TO_DWORD((CIRD01.OnDelay)/60/1000));
				TxLen:=TxLen+RAWTOHEX(ADR(j),2,ADR(TxData[TxLen]));
				j:=DWORD_TO_WORD(TIME_TO_DWORD((CIR01.OffDelay)/60/1000));
				TxLen:=TxLen+RAWTOHEX(ADR(j),2,ADR(TxData[TxLen]));

		END_CASE


	6: (* LEGGO ALLARME PRESENTE SUL CIRCOLATORE *)
		Cmd_RLen:=2;
			CASE Cmd_ObjIdx OF
			1:	j:=(CIRD01.DataPump1.PumpAlarm[0]);
				TxLen:=TxLen+RAWTOHEX(ADR(j),2,ADR(TxData[TxLen]));
				j:=(CIRD01.DataPump2.PumpAlarm[0]);
				TxLen:=TxLen+RAWTOHEX(ADR(j),2,ADR(TxData[TxLen]));

		END_CASE



ELSE
	Cmd_R:=3;
END_CASE

*)
END_ACTION
ACTION Cmd_CRON:
(* Check index *)
IF Cmd_ObjIdx<1 OR Cmd_ObjIdx>250 THEN
	Cmd_R:=2;
	RETURN;
END_IF

(* Process command *)
CASE Cmd_C OF

	1: (* GET PROFILE *)
		IF Cmd_CLen<>3 THEN
			Cmd_R:=4;
		ELSE
			(* Load profile *)
			CronEd.CN_Sel:=WORD_TO_BYTE(Cmd_ObjIdx);
			Cmd_Buf_U16:=ADR(Cmd_Buf[8]);
			CronEd.CN_YSel:=Cmd_Buf_U16^;
			IF Cmd_Buf[10]<=10 THEN
				CronEd.PR_Sel:=Cmd_Buf[10];
				CronEd.PR_Load_Exe();
				(* Response data *)
				Cmd_RLen:=DOUBLE_MIN_FOR_DAY;		(*192;  *)
				TxLen:=TxLen+RAWTOHEX(ADR(CronEd.PR.Setpoint),DOUBLE_MIN_FOR_DAY ,ADR(TxData[TxLen]));
			ELSE
				Cmd_R:=6;
			END_IF
		END_IF

	2: (* SET PROFILE *)
		IF Cmd_CLen<>(3+DOUBLE_MIN_FOR_DAY) THEN
			Cmd_R:=4;
		ELSE
			(* Save profile *)
			CronEd.CN_Sel:=WORD_TO_BYTE(Cmd_ObjIdx);
			Cmd_Buf_U16:=ADR(Cmd_Buf[8]);
			CronEd.CN_YSel:=Cmd_Buf_U16^;
			IF Cmd_Buf[10]<=10 THEN
				CronEd.PR_Sel:=Cmd_Buf[10];
				MEMCPY(ADR(Cmd_Buf[11]),ADR(CronEd.PR.Setpoint),DOUBLE_MIN_FOR_DAY);		(* DOUBLE_MIN_FOR_DAY *)
				CronEd.PR_Save_Exe();
				Cmd_RLen:=0;
			ELSE
				Cmd_R:=6;
			END_IF
		END_IF

	5: (* GET CALENDAR MONTH *)
		IF Cmd_CLen<>3 THEN
			Cmd_R:=4;
		ELSE
			(* Load calendar *)
			CronEd.CN_Sel:=WORD_TO_BYTE(Cmd_ObjIdx);
			Cmd_Buf_U16:=ADR(Cmd_Buf[8]);
			CronEd.CN_YSel:=Cmd_Buf_U16^;
			IF Cmd_Buf[10]>=1 AND Cmd_Buf[10]<=12 THEN
				CronEd.CA_Sel:=Cmd_Buf[10];
				CronEd.CA_Load_Exe();
				(* Response data *)
				Cmd_RLen:=32;
				TxLen:=TxLen+RAWTOHEX(ADR(CronEd.CA.Profile),32,ADR(TxData[TxLen]));
			ELSE
				Cmd_R:=6;
			END_IF
		END_IF

	6: (* SET CALENDAR MONTH *)
		IF Cmd_CLen<>(3+32) THEN
			Cmd_R:=4;
		ELSE
			(* Save calendar *)
			CronEd.CN_Sel:=WORD_TO_BYTE(Cmd_ObjIdx);
			Cmd_Buf_U16:=ADR(Cmd_Buf[8]);
			CronEd.CN_YSel:=Cmd_Buf_U16^;
			IF Cmd_Buf[10]>=1 AND Cmd_Buf[10]<=12 THEN
				CronEd.CA_Sel:=Cmd_Buf[10];
				MEMCPY(ADR(Cmd_Buf[11]),ADR(CronEd.CA.Profile),32);
				CronEd.CA_Save_Exe();
			ELSE
				Cmd_R:=6;
			END_IF
		END_IF

	9: (* CRON RESTART *)
		IF Cmd_ObjIdx>=1 AND Cmd_ObjIdx <=CRON_MAX THEN
			CRON[Cmd_ObjIdx].InitOK:=FALSE;
		END_IF


ELSE
	Cmd_R:=3;
END_CASE
END_ACTION
ACTION Cmd_CTL:
RETURN;
(*
IF Cmd_ObjIdx<1 OR Cmd_ObjIdx>3 THEN
	Cmd_R:=2;
	RETURN;
END_IF

(* Process command *)
CASE Cmd_C OF

	0:	(* Comando limiti contalitri *)
		CASE Cmd_ObjIdx OF

		1: (* Scrittura Limite accettabile di pedite *)
			Cmd_Buf_U16:=ADR(Cmd_Buf[8]);
			CTL01.LimiteMaxPerdita:= Cmd_Buf_U16^;


		2: (* Scrittura Limite accettabile di pedite *)
			Cmd_Buf_U16:=ADR(Cmd_Buf[8]);
			CTL02.LimiteMaxPerdita:= Cmd_Buf_U16^;

		3: (* Scrittura Limite accettabile di pedite *)
			Cmd_Buf_U16:=ADR(Cmd_Buf[8]);
			CTL03.LimiteMaxPerdita:= Cmd_Buf_U16^;
		END_CASE

ELSE
	Cmd_R:=3;
END_CASE
 *)
END_ACTION
ACTION Cmd_GRU:
RETURN;
(* Check index *)
(*
IF Cmd_ObjIdx<>1 THEN
	Cmd_R:=2;
	RETURN;
END_IF

(* Process command *)
CASE Cmd_C OF

	1: (* GET CLIMATIC *)
		Cmd_RLen:=20;
		FOR i:=0 TO 4 DO
			j:=DINT_TO_INT(GRU01_Clima.Points[i].X);
			TxLen:=TxLen+RAWTOHEX(ADR(j),2,ADR(TxData[TxLen]));
			j:=DINT_TO_INT(GRU01_Clima.Points[i].Y);
			TxLen:=TxLen+RAWTOHEX(ADR(j),2,ADR(TxData[TxLen]));
		END_FOR

	2: (* SET CLIMATIC *)
		IF Cmd_CLen<>20 THEN
			Cmd_R:=4;
		ELSE
			FOR i:=0 TO 4 DO
				Cmd_Buf_INT:=ADR(Cmd_Buf[8+4*i]); j:=Cmd_Buf_INT^;
				GRU01_Clima.Points[i].X:=INT_TO_DINT(j);
				Cmd_Buf_INT:=ADR(Cmd_Buf[10+4*i]); j:=Cmd_Buf_INT^;
				GRU01_Clima.Points[i].Y:=INT_TO_DINT(j);
			END_FOR
		END_IF

ELSE
	Cmd_R:=3;
END_CASE
 *)
END_ACTION
ACTION Cmd_Lux:
(* Check index *)
IF Cmd_ObjIdx<1 OR Cmd_ObjIdx>MAX_LUXNUM THEN
	Cmd_R:=2; (* id del lux fuori range *)
	RETURN;
END_IF
(*
x:=1;
WHILE (Cmd_ObjIdx <> TabDefaultLux[x].LuxNumber) AND ( x <= MAX_LUXNUM) DO
	x := x + 1;
END_WHILE
 *)
(*
IF Cmd_ObjIdx = TabDefaultLux[x].LuxNumber THEN
*)

x:=Cmd_ObjIdx;
	(* Process command *)
	CASE Cmd_C OF

		0:	(* Restore default functioning mode *)
		LuxElement[x].CTRL_MODE:=LuxElement[x].CTRL_MODE_backUp;
		LuxElement[x](LocalWorkingTime:=GlobalWorkingtime[x],LocalPowerOnCycles:=GlobalPowerOnCycles[x],
													LocalEnergyCounter:=GlobalEnergyCounter[x],
													LocalEnergyCounter_t:=GlobalEnergyCounter_t[x]);

		1:	(* Reset statistic counter *)
		LuxElement[x].StatReset(LocalWorkingTime:=GlobalWorkingtime[x],LocalPowerOnCycles:=GlobalPowerOnCycles[x],
													LocalEnergyCounter:=GlobalEnergyCounter[x],
													LocalEnergyCounter_t:=GlobalEnergyCounter_t[x]);

		2,3:	(* Switch On (command=2) or Off (command=3) lux *)
		CASE Cmd_C OF
			2: (*switch a Manuale ON*)
			LuxElement[x].CTRL_MODE := 1; (* Set TO manuale ON  *)
			LuxElement[x](LocalWorkingTime:=GlobalWorkingtime[x],LocalPowerOnCycles:=GlobalPowerOnCycles[x],
													LocalEnergyCounter:=GlobalEnergyCounter[x],
													LocalEnergyCounter_t:=GlobalEnergyCounter_t[x]);
			3: (*switch a Manuale OFF*)
			LuxElement[x].CTRL_MODE := 0; (* Set TO manuale OFF  *)
			LuxElement[x](LocalWorkingTime:=GlobalWorkingtime[x],LocalPowerOnCycles:=GlobalPowerOnCycles[x],
													LocalEnergyCounter:=GlobalEnergyCounter[x],
													LocalEnergyCounter_t:=GlobalEnergyCounter_t[x]);

		END_CASE
		4: (* Modify timer value *)
	(*	IF TabDefaultLux[x].Mode = 03 THEN  la modifica ha senso per i lux a timer  *)
		IF LuxElement[x].CTRL_MODE = 03 THEN (* la modifica ha senso per i lux a timer  *)
			NewValueTimerH:=BYTE_TO_WORD(Cmd_Buf[8]);
			NewValueTimerH:=SHL(NewValueTimerH,8);
			NewValueTimerH:=NewValueTimerH+BYTE_TO_WORD(Cmd_Buf[9]);
			(*  NewValueTimerH:=ROL(NewValueTimerH, 8);   *)

			NewValueTimerL:=BYTE_TO_WORD(Cmd_Buf[10]);
			NewValueTimerL:=SHL(NewValueTimerL,8);
			NewValueTimerL:=NewValueTimerL+BYTE_TO_WORD(Cmd_Buf[11]);
			(* NewValueTimerL:=ROL(NewValueTimerL, 8);  *)

			NewValueTimer:=WORD_TO_DWORD(NewValueTimerH);
			NewValueTimer:=SHL(NewValueTimer,16);
			NewValueTimer:=NewValueTimer+WORD_TO_DWORD(NewValueTimerL);
			IF NewValueTimer>4294966 THEN
				Cmd_R:=3; (* Comando errato valore timer overflow		 *)

(*
			NewValueTimer:=byte_to_dword(Cmd_Buf[8]);
			NewValueTimer:=SHL(NewValueTimer,8); 
			NewValueTimer:=NewValueTimer+byte_to_dword(Cmd_Buf[9]);
			NewValueTimer:=SHL(NewValueTimer,8); 
			NewValueTimer:=NewValueTimer+byte_to_dword(Cmd_Buf[10]);
			NewValueTimer:=SHL(NewValueTimer,8); 
			NewValueTimer:=NewValueTimer+byte_to_dword(Cmd_Buf[11]);
*)
(*
			ELSE
					TabLuxPsg[x].TimerOn := DWORD_TO_TIME(NewValueTimer*1000);
				FOR x := 1 TO MAX_LUXNUM DO
					IF LuxElement[x].ID = Cmd_ObjIdx
						THEN LuxElement[x].LuxTimer := DWORD_TO_TIME(NewValueTimer*1000);  (*  set del nuovo valore del timer del lux 	 *)
					END_IF
				END_FOR
*)
			END_IF
		ELSE
			Cmd_R:=3; (* Comando errato / non previsto *)
		END_IF
		5:	(* get working mode*)
			Cmd_RLen:=2;
			ModeFromPlc:=LuxElement[x].CTRL_MODE;
			(* ModeFromPlc:=ROL(ModeFromPlc, 8);  *)
			TxLen:=TxLen+RAWTOHEX(ADR(ModeFromPlc),2,ADR(TxData[TxLen]));


(*		6:  Modify dimming value for timer control *)
(*		7:  Modify dimming value for key control *)
(*		8:  Modify start and stop orari di funzionamento dei lux a timer *)

	ELSE
		Cmd_R:=3;  (*  Comando errato / non previsto *)
	END_CASE

(*
ELSE
	Cmd_R:=2; (* id del lux non presente in lista *)
END_IF
*)
END_ACTION
ACTION Cmd_PDC:
;(* Check index *)(*
IF Cmd_ObjIdx<>1 THEN
	Cmd_R:=2;
	RETURN;
END_IF

(* Process command *)
CASE Cmd_C OF

	3: (* TRY REARM *)
		PDC01.Rearm:=TRUE;

ELSE
	Cmd_R:=3;
END_CASE
*);
END_ACTION
ACTION Cmd_SYS:
(* Check index *)
IF Cmd_ObjIdx<>0 THEN
	Cmd_R:=2;
	RETURN;
END_IF

(* Process command *)
CASE Cmd_C OF

	0: (* ECHO *)
		IF Cmd_CLen<>0 THEN
			TxLen:=0;
		END_IF

	1: (* LOG REQUEST *)
		LogTrig();

	2: (* REARM *)
		Sys.Warning:=FALSE;
		Sys.Alarm:=FALSE;
		Sys.AlarmStop:=FALSE;

	3: (* GET INFO1 *)
		Cmd_RLen:=6;
		TxLen:=TxLen+RAWTOHEX(ADR(Plant_SN),4,ADR(TxData[TxLen]));
		TxLen:=TxLen+RAWTOHEX(ADR(Plant_SW_VER),2,ADR(TxData[TxLen]));

	4: (*  Scrivo i Parametri gestione Impianto   *)

			Cmd_Buf_U16:=ADR(Cmd_Buf[8]);
			DelayAllarmeTemperaturaNonRaggiunta := Cmd_Buf_U16^; 			(* Ritardo Allarme dall'avvio Caldaia*)
			Cmd_Buf_U16:=ADR(Cmd_Buf[10]);
			DeltaInterventoAllarmeTempeaturaNonRaggiuta := Cmd_Buf_U16^;	(* Delta Soglia Temperatura per Allarme Temperatura Non Raggiunta *)
			Cmd_Buf_U16:=ADR(Cmd_Buf[12]);
			OffsetSetPointManuale := Cmd_Buf_U16^; 					(* Offest Perdite Scambiatore  *)

	5: (*  Leggi i parametri gestione Impianto  *)

			Cmd_RLen:=14;
			j:=(DelayAllarmeTemperaturaNonRaggiunta);   				(* Ritardo Allarme dall'avvio Caldaia*)
			TxLen:=TxLen+RAWTOHEX(ADR(j),2,ADR(TxData[TxLen]));
			j:=(DeltaInterventoAllarmeTempeaturaNonRaggiuta);			(* Delta Soglia Temperatura per Allarme Temperatura Non Raggiunta *)
			TxLen:=TxLen+RAWTOHEX(ADR(j),2,ADR(TxData[TxLen]));
			j:=(OffsetSetPointManuale);									(* Offest Perdite Scambiatore  *)
			TxLen:=TxLen+RAWTOHEX(ADR(j),2,ADR(TxData[TxLen]));

	6: (*  Scrivo i Parametri gestione Impianto - Antigelo   *)

			Cmd_Buf_U16:=ADR(Cmd_Buf[8]);
			SogliaMinStartAntigelo := Cmd_Buf_U16^; 			(* Soglia mininma Start Antigelo *)
			Cmd_Buf_U16:=ADR(Cmd_Buf[10]);
			SogliaMinStopAntigelo := Cmd_Buf_U16^;				(* Soglia Massima Stop Antigelo *)
			Cmd_Buf_U16:=ADR(Cmd_Buf[12]);
			BitAbilitaAntigelo :=INT_TO_BOOL( Cmd_Buf_U16^); 	(* Abilitazione Antigelo  *)

	7: (*  Leggi i parametri gestione Impianto - Antigelo *)

			Cmd_RLen:=14;
			j:=(SogliaMinStartAntigelo); 							(* Soglia mininma Start Antigelo *)
			TxLen:=TxLen+RAWTOHEX(ADR(j),2,ADR(TxData[TxLen]));
			j:=(SogliaMinStopAntigelo);								(* Soglia Massima Stop Antigelo *)
			TxLen:=TxLen+RAWTOHEX(ADR(j),2,ADR(TxData[TxLen]));
			j:=BOOL_TO_INT(BitAbilitaAntigelo);						(* Abilitazione Antigelo  *)
			TxLen:=TxLen+RAWTOHEX(ADR(j),2,ADR(TxData[TxLen]));

	14: (*  Imposto data e ora del PLC  *)


			Cmd_Buf_U16:=ADR(Cmd_Buf[8]);
			SetAnno:= Cmd_Buf_U16^; 												(* Anno *)
			Cmd_Buf_U16:=ADR(Cmd_Buf[10]);
			SetMese:= Cmd_Buf_U16^;												 	(* mese *)
			Cmd_Buf_U16:=ADR(Cmd_Buf[12]);
			SetGiorno:=( Cmd_Buf_U16^);											 	(* Giorno *)
			Cmd_Buf_U16:=ADR(Cmd_Buf[14]);
			SetOra:=( Cmd_Buf_U16^); 												(* ora *)
			Cmd_Buf_U16:=ADR(Cmd_Buf[16]);
			SetMinuti:= ( Cmd_Buf_U16^);										 	(* Minuti *)
			Cmd_Buf_U16:=ADR(Cmd_Buf[18]);
			SetSecondi:= ( Cmd_Buf_U16^);										 	(* secondi *)

	(*		SysRtcSetTime(SetDataTime(DWORD_TO_INT(ADR(Cmd_Buf[8])),				(* Anno *)
										DWORD_TO_INT(ADR(Cmd_Buf[10])),				(* mese *)
										DWORD_TO_INT(ADR(Cmd_Buf[11])),				(* Giorno *)
										DWORD_TO_INT(ADR(Cmd_Buf[12])),				(* ora *)
										DWORD_TO_INT(ADR(Cmd_Buf[13])),				(* Minuti *)
										DWORD_TO_INT(ADR(Cmd_Buf[14]))				(* secondi *)
										)); *)

		SysRtcSetTime((SetDataTime(SetAnno,SetMese,SetGiorno,SetOra,SetMinuti,SetSecondi)));





ELSE
	Cmd_R:=3;
END_CASE
END_ACTION
ACTION Cmd_VRD:
RETURN;
(* Check index *)
(*
IF Cmd_ObjIdx<1 OR Cmd_ObjIdx>3 THEN
	Cmd_R:=2;
	RETURN;
END_IF

(* Process command *)
CASE Cmd_C OF

	1: (* GET CLIMATIC *)
		Cmd_RLen:=20;
		FOR i:=0 TO 4 DO
			IF Cmd_ObjIdx=1 THEN
				j:=DINT_TO_INT(VRD01_Clima.Points[i].X);
			END_IF
			IF Cmd_ObjIdx=2 THEN
				j:=DINT_TO_INT(VRD02_Clima.Points[i].X);
			END_IF
			IF Cmd_ObjIdx=3 THEN
				j:=DINT_TO_INT(VRD03_Clima.Points[i].X);
			END_IF
			TxLen:=TxLen+RAWTOHEX(ADR(j),2,ADR(TxData[TxLen]));
			IF Cmd_ObjIdx=1 THEN
				j:=DINT_TO_INT(VRD01_Clima.Points[i].Y);
			END_IF
			IF Cmd_ObjIdx=2 THEN
				j:=DINT_TO_INT(VRD02_Clima.Points[i].Y);
			END_IF
			IF Cmd_ObjIdx=3 THEN
				j:=DINT_TO_INT(VRD03_Clima.Points[i].Y);
			END_IF
			TxLen:=TxLen+RAWTOHEX(ADR(j),2,ADR(TxData[TxLen]));
		END_FOR

	2: (* SET CLIMATIC *)
		IF Cmd_CLen<>20 THEN
			Cmd_R:=4;
		ELSE
			FOR i:=0 TO 4 DO
				Cmd_Buf_INT:=ADR(Cmd_Buf[8+4*i]); j:=Cmd_Buf_INT^;
				IF Cmd_ObjIdx=1 THEN
					VRD01_Clima.Points[i].X:=INT_TO_DINT(j);
				END_IF
				IF Cmd_ObjIdx=2 THEN
					VRD02_Clima.Points[i].X:=INT_TO_DINT(j);
				END_IF
				IF Cmd_ObjIdx=3 THEN
					VRD03_Clima.Points[i].X:=INT_TO_DINT(j);
				END_IF
				Cmd_Buf_INT:=ADR(Cmd_Buf[10+4*i]); j:=Cmd_Buf_INT^;
				IF Cmd_ObjIdx=1 THEN
					VRD01_Clima.Points[i].Y:=INT_TO_DINT(j);
				END_IF
				IF Cmd_ObjIdx=2 THEN
					VRD02_Clima.Points[i].Y:=INT_TO_DINT(j);
				END_IF
				IF Cmd_ObjIdx=3 THEN
					VRD03_Clima.Points[i].Y:=INT_TO_DINT(j);
				END_IF

			END_FOR
		END_IF

ELSE
	Cmd_R:=3;
END_CASE

 *)
END_ACTION
ACTION Command:
(* Default response OK/NODATA *)
Cmd_R:=0;
Cmd_RLen:=0;
TxLen:=16;

(* Check object *)
CASE Cmd_Obj OF

	EO_SYS:
		Cmd_SYS();

	EO_LUX:
		Cmd_LUX();

	EO_CRON:
		Cmd_CRON();

ELSE
	Cmd_R:=3;
END_CASE

(* Generate response *)
IF TxLen>0 THEN
	RAWTOHEX(ADR(Cmd_Obj)	,2,ADR(TxData[ 0]));
	RAWTOHEX(ADR(Cmd_ObjIdx),2,ADR(TxData[ 4]));
	RAWTOHEX(ADR(Cmd_R)		,2,ADR(TxData[ 8]));
	RAWTOHEX(ADR(Cmd_RLen)	,2,ADR(TxData[12]));
	TxTrig:=TRUE;
END_IF
END_ACTION

(* POU Utils Functions/TCPSERVER, ST *)
FUNCTION_BLOCK TCPSERVER
(***********************************************************************************************************	*)
(* Version: 1.6                                    			          											*)
(* Date: 11.02.2011                                   					          							    *)
(***********************************************************************************************************	*)
(* WAGO Kontakttechnik GmbH Hansastr. 27 32423 Minden(Westf.)													*)
(* Tel. +0049 571/887-0 Fax. +0049 571/887-0																	*)
(* Author: VB																									*)
(***********************************************************************************************************	*)
(*Description:	A TCP server to read and write data													       		*)
(*Historie:																										*)
(*Version 1.6: 11.02.2011: Changes according to 750-880/881											 			*)
(*Version 1.5: 27.11.2008 Bugfix allow reuse port																*)
(*Version 1.4: 13.10.2008 Bugfix transmitting large data														*)
(*Version 1.3: 15.01.2007 Changes according to FW11																*)
(*Version 1.2: 09.03.2006 Changes for socket handle 0											       			*)
(*Version 1.1: 14.02.2005 Release																				*)
(***********************************************************************************************************	*)
VAR CONSTANT
	STATE_INIT     				 : BYTE:= 0;
	STATE_OPEN     				 : BYTE:= 1;
	STATE_TX       				 : BYTE:= 20;
	STATE_RX       				 : BYTE:= 30;
	STATE_CLOSE    				 : BYTE:= 40;
	STATE_ERROR_TRAP		 	 : BYTE:= 200;
END_VAR
VAR_INPUT
	xEnable    					: BOOL;	 (* Set TRUE to enable function block *)
	wPortNumber					: WORD;  (* Port *)
	tServerTimeOut				: TIME:=t#50s;
	ptSendData					: POINTER TO ARRAY[0..MAX_SEND_TCP_SERVER] OF BYTE;
	diSendCount					: DINT;
END_VAR
VAR_OUTPUT
	xClientConnected  			: BOOL:= FALSE;
	diError 					: DINT:= 0;
END_VAR
(* Status Codes -----------------------------------------
	16#8001 => No socket descriptor available 
	16#8002 => SysSockBind fails 
	16#8003 => SysSockListen fails 
	16#8004 => switching to none blocking mode fails
	16#8005 => SysSockClose() returns FALSE 
    16#8006 => SysSockConnect() fails
    16#8007 => SysSockSend() fails
	16#8008 => error state machine 
	16#8009 => timeout while waiting for data from server 
	16#0001 => server waiting for client to establish connection
------------------------------------------------------------*)
VAR_IN_OUT
	xStartSend					: BOOL;
	aReceiveBuffer				: ARRAY [0..MAX_RECEIVE_TCP_SERVER] OF BYTE;
	diReceiveCount				: DINT;
END_VAR

VAR
	m_State    					: BYTE:= 0;
	m_ReceiveBuffer				: ARRAY [0..MAX_RECEIVE_TCP_SERVER_SOCKET] OF BYTE;
	m_ServerSocket				: DINT:= SOCKET_INVALID;
	m_Socket					: DINT:= SOCKET_INVALID;
	m_AddressInfo				: SOCKADDRESS;
	m_BytesReceived				: DINT;
	m_diReturn					: DINT;
	m_xReturn					: BOOL;
	m_SizeSockadr				: DWORD;
	m_ConnectionWatchdog		: TON;
	m_Flags						: DINT;
	m_NoneBlocking   			: DINT:= 1;
	m_Blocking   				: DINT:= 0;
	i							: INT;
	m_count						: DINT;
	diOption					: DINT := 1;
	on: DINT;
END_VAR
IF xEnable THEN
	CASE m_State OF
		STATE_INIT:
			(* Create Socket *)
			m_ServerSocket:= SysSockCreate( SOCKET_AF_INET, SOCKET_STREAM, 0);
			IF m_ServerSocket = SOCKET_INVALID THEN
				(* *)
				diError:= 16#8001;
				m_State:= STATE_ERROR_TRAP;
				RETURN;
			ELSE
				;
			END_IF
			(* Address bindings *)
			(********************)
			on:=1;
			SysSockSetOption( m_ServerSocket, SOCKET_SOL, SOCKET_SO_REUSEADDR, ADR(on), SIZEOF(on) );

			m_AddressInfo.sin_family:= SOCKET_AF_INET;
			m_AddressInfo.sin_port  := SysSockHtons( wPortNumber);
			m_AddressInfo.sin_addr  := SOCKET_INADDR_ANY;
			IF NOT SysSockBind( m_ServerSocket, ADR(m_AddressInfo), SIZEOF(m_AddressInfo)) THEN
				diError:= 16#8002;
				m_State:= STATE_ERROR_TRAP;
				RETURN;
			END_IF
			(* Wait for connections *)
			(************************)
			IF NOT SysSockListen( m_ServerSocket, 1) THEN
				diError:= 16#8003;
				m_State:= STATE_ERROR_TRAP;
			END_IF

			(* Puts SOCKET in NonBlocking mode *)
			m_diReturn:= SysSockIoctl( m_ServerSocket, SOCKET_FIONBIO, ADR(m_NoneBlocking));

			m_State:= STATE_OPEN;


		STATE_OPEN: 	(* Waiting for incomming connection *)
				m_SizeSockadr:=SIZEOF(m_AddressInfo);
				m_Socket:= SysSockAccept( m_ServerSocket, ADR(m_AddressInfo), ADR(m_SizeSockadr));
				diError:=State_open;
				IF m_Socket <> SOCKET_INVALID THEN
					xClientConnected:=TRUE;
					(*Set Push-Bit:new V1.5*)
					IF ADR(%MW0)=16#30000000  OR ADR(%MW0)=16#20000000 THEN (*841 or 881*)
						SysSockSetOption(
							diSocket:=m_Socket,
							diLevel:=6,
							diOption:=SOCKET_TCP_NODELAY,
							pOptionValue:=ADR(diOption),
							diOptionLength:=SIZEOF(diOption));
					ELSE
							;
					END_IF
					SysSockIoctl( m_Socket, SOCKET_FIONBIO, ADR(m_NoneBlocking));
					m_State:= STATE_RX;
					diError:=0;
				END_IF

		STATE_RX:
					m_BytesReceived:= SysSockRecv( m_Socket, ADR(m_ReceiveBuffer), SIZEOF(m_ReceiveBuffer), 0);
					CASE m_BytesReceived OF
					-1:(*no data available or error occured*)
						m_ConnectionWatchdog(IN:=TRUE , PT:=tServerTimeOut );
						IF m_connectionWatchdog.Q THEN
							m_State:= STATE_CLOSE;
							m_ConnectionWatchdog(IN:=FALSE);(*reset connection watchdog*)
							diError := 16#8009;
						END_IF
					0:(* socket was "gracefully closed"  *)
						m_State:= STATE_CLOSE;
						diError := 16#8003;
					ELSE
						(* Copy received data into receive buffer *)
						(********************************)
						FOR i:= 0 TO DINT_TO_INT(m_BytesReceived	)-1 DO
							aReceiveBuffer[diReceiveCount]:= m_ReceiveBuffer[i];
							diReceiveCount:=(diReceiveCount+1) MOD SIZEOF(aReceiveBuffer);
						END_FOR

						m_ConnectionWatchdog(IN:=FALSE);(*reset connection watchdog*)
					END_CASE

				(*send data*)
				IF xStartSend	 THEN
					m_State := STATE_TX;
				END_IF

	STATE_TX:	 (* send TCP-message *)
		m_diReturn := SysSockSend(diSocket := m_Socket,
								  pbyBuffer := ADR(ptSendData^[m_count]),(*geändert V1.4 bisher: [0] *)
								  diBufferSize := diSendCount-m_count,
								  diFlags :=m_Flags);
		CASE m_diReturn OF
		-1:	(* ERROR or data could not yet be send (V1.3 due to new FW11) *)
			m_ConnectionWatchdog(IN:=TRUE , PT:=tServerTimeOut );
			IF m_connectionWatchdog.Q THEN
				m_State:= STATE_CLOSE;
				m_ConnectionWatchdog(IN:=FALSE);(*reset connection watchdog*)
				diError := 16#8007;
			END_IF
		0: (* socket was "gracefully closed"  *)
			m_State := STATE_CLOSE;
			diError := 16#8003;
		ELSE (* succesful *)
			m_count:=m_count+m_diReturn;
			IF m_count>=diSendCount THEN
				diError := 16#0000;
				m_State := STATE_RX;
				m_count:=0;
				xStartSend:=FALSE;
			END_IF
			m_ConnectionWatchdog(IN:=FALSE);(*reset connection watchdog*)
		END_CASE


		STATE_CLOSE:	(* Close the server *)

		IF ADR(%MW0)=16#30000000  OR ADR(%MW0)=16#20000000 THEN (*841 or 881*)
			;
		ELSE
			IF m_Socket>=0 THEN
				SysSockShutdown(m_Socket, 0);;(*870*)
			END_IF
		END_IF
		IF m_Socket>=0 THEN
			SysSockClose( m_Socket);
		END_IF
		xClientConnected:= FALSE;
		m_State:= STATE_OPEN; (* Try to open the server again *)
		m_ConnectionWatchdog(IN:=FALSE);(*reset connection watchdog*)

		STATE_ERROR_TRAP: (* Error Read/Write socket  *)
			m_State:= STATE_ERROR_TRAP;

	ELSE  (* Bad FSM code trap  *)
			m_State:= STATE_ERROR_TRAP;
			diError:= 16#8008;
	END_CASE;
ELSE
	IF m_State <> STATE_INIT THEN
		IF ADR(%MW0)=16#30000000  OR ADR(%MW0)=16#20000000 THEN (*841 or 881*)
			;
		ELSE
			IF m_Socket>=0 THEN
				SysSockShutdown(m_Socket, 0);;(*870*)
			END_IF
		END_IF
		IF m_Socket>=0 THEN
			SysSockClose( m_Socket);
		END_IF
		IF ADR(%MW0)=16#30000000  OR ADR(%MW0)=16#20000000 THEN (*841 or 881*)
			;
		ELSE
			IF m_ServerSocket>=0 THEN
				SysSockShutdown(m_ServerSocket, 0);;(*870*)
			END_IF
		END_IF
		IF m_ServerSocket>=0 THEN
			SysSockClose( m_ServerSocket);
		END_IF
		xClientConnected:= FALSE;
		diError:= 0;
		m_State:= STATE_init; (* Try to open the server again *)
		m_ConnectionWatchdog(IN:=FALSE);(*reset connection watchdog*)
	END_IF
END_IF
END_FUNCTION_BLOCK

(* POU Utils Functions/HEXTORAW, ST *)
FUNCTION HEXTORAW : WORD
VAR_INPUT
	pString		: POINTER TO BYTE;
	StringLen	: WORD;
	pData		: POINTER TO BYTE;
END_VAR
VAR
	xl: WORD;
	xi: WORD;
	xr: BYTE;
END_VAR
xl:=0;
xi:=0;

WHILE xi<StringLen DO

	IF pString^>=97 AND pString^<=102 THEN
		xr := pString^ - 87;
	ELSIF pString^>=65 AND pString^<=70 THEN
		xr := pString^ - 55;
	ELSIF pString^>=48 AND pString^<=57 THEN
		xr := pString^ - 48;
	ELSE
		xr := 16;
	END_IF

	IF xr<16 THEN
		IF (xi AND 1)=0 THEN
			pData^ := xr * 16;
		ELSE
			pData^ := pData^ + xr;
			pData := pData + 1;
			xl := xl + 1;
		END_IF
	END_IF

	xi := xi + 1;
	pString := pString + 1;

END_WHILE

HEXTORAW:=xl;
END_FUNCTION

(* POU Utils Functions/RAWTOHEX, ST *)
FUNCTION RAWTOHEX : WORD
VAR_INPUT
	pData: POINTER TO BYTE;
	DataLen: WORD;
	pString: POINTER TO BYTE;
END_VAR
VAR
	xl: WORD;
END_VAR
xl:=0;

WHILE DataLen>0 DO

	pString^ := (pData^ / 16#10) + 48 + (((pData^ / 16#10)/10)*7);
	pString:=pString+1;
	pString^ := (pData^ AND 16#0F)  + 48 + (((pData^ AND 16#0F)/10)*7);
	pString:=pString+1;
	pData:=pData+1;
	DataLen:=DataLen-1;
	xl:=xl+2;

END_WHILE

(*pString^:=0;*)

RAWTOHEX:=xl;
END_FUNCTION

(* POU Utils Functions/GestioneDataTime_DaOscat/SetDataTime, ST *)
FUNCTION SetDataTime : DT
VAR_INPUT
	year : INT;
	month : INT;
	day : INT;
	hour : INT;
	minute : INT;
	second : INT;
END_VAR

VAR
	count : INT;
END_VAR
(* Creazione variabiletipo DT per creare Orario da dare al PLC *)


IF month > 2 THEN
	count := (month - 1) * 30;
	IF month > 7 THEN count := count + SHR(month - 3,1); ELSE count := count + SHR(month - 4,1); END_IF;
	(* chech for leap year and add one day if true *)
	IF SHL(year,14) = 0 THEN count := count + 1; END_IF;
ELSE
	count := (month - 1) * 31;
END_IF;


SetDataTime := DWORD_TO_DT(DATE_TO_DWORD( DWORD_TO_DATE((INT_TO_DWORD(count + day - 1) + SHR(INT_TO_DWORD(year) * 1461 - 2878169, 2)) * 86400))
				+ INT_TO_DWORD(SECOND)
				+ INT_TO_DWORD(MINUTE) * 60
				+ INT_TO_DWORD(HOUR) * 3600);
END_FUNCTION

(* POU Configuration/MODBUS_CONFIGURATION, ST *)
PROGRAM MODBUS_CONFIGURATION        
VAR                                
END_VAR                            
(*                                 
   <?xml version="1.0" encoding="UTF-16" standalone="yes"?>
<network xml_structure_version="1" xml_feature_version="1">
	<generator_settings minRTUTaskCycleTimeMs="5" minEthaskCycleTimeMs="5" ethSlaveMultiplier="0.1" rtuInterfaceMultiplier="0.1" taskGeneration="false"/>
</network>
                              
*)                                 
;                                  
END_PROGRAM

(* POU Plant/SYS_Proc, ST *)
PROGRAM SYS_Proc
VAR
(*	fALARM_PB		:FLT_TAP;
	fALARM_TB		:FLT_TAP;
	fALARM_PM		:FLT_TAP;	*)

(*	fGZB_ST			:FLT_TAP;  (* GATEWAY ZIGBEE *)*)
(*	fVPN_ST1		:FLT_TAP;  (* VPN CONNECT *)*)
	fVPN_ST2		:FLT_TAP;  (* VPN STATUS *)
(*	fKEY_CT_ST		:FLT_TAP;  (* DOOR1 *)*)
(*	fKEY_SCT_ST		:FLT_TAP;  (* DOOR2 *)*)
	fKEY_QE_ST		:FLT_TAP;  (* DOOR3 *)


	fBostAttivo	:FLT_TAP;

	fALARM_MancatoRaggiungimentoAcqua		:FLT_TAP;
	DelayfALARM_MancatoRaggiungimentoAcqua:TON;



END_VAR
(*************** ISPESL *****************)
RETURN;

(*fALARM_PB(IN:=ALARM_PB);
IF fALARM_PB.EVH THEN
	LogEv(EL_AlarmStop,EO_PBV,1,1,'Over_Pressure_Alarm');
END_IF

fALARM_TB(IN:=ALARM_TB);
IF fALARM_TB.EVH THEN
	LogEv(EL_AlarmStop,EO_TBV,1,1,'Over_Temperature_Alarm');
END_IF

fALARM_PM(IN:=ALARM_PM);
IF fALARM_PM.EVH THEN
	LogEv(EL_AlarmStop,EO_PMV,1,1,'Under_Pressure_Alarm');
END_IF
*)
(****************************************)

(*### VPN Connection Check ###*)(*
fVPN_ST1(IN:=VPN_ST1);
IF fVPN_ST1.EVH THEN
	LogEv(EL_Log,EO_VPN,1,1,'CONNECT_ON');
END_IF
IF fVPN_ST1.EVL THEN
	LogEv(EL_Log,EO_VPN,1,2,'CONNECT_OFF');
END_IF*)

(*### VPN Status Check ###*)
(*
fVPN_ST2(IN:=VPN_ST2);
IF fVPN_ST2.EVH THEN
	LogEv(EL_Log,EO_VPN,1,3,'STATUS_UP');
END_IF
IF fVPN_ST2.EVL THEN
	LogEv(EL_Wrn,EO_VPN,1,4,'STATUS_DOWN');
END_IF
*)
(*### DOOR01 Status Check ###*)(*
fKEY_CT_ST(IN:=KEY_CT_ST);
IF fKEY_CT_ST.EVH THEN
	LogEv(EL_Log,EO_DOOR,1,2,'Centrale_termica_Close');
END_IF
IF fKEY_CT_ST.EVL THEN
	LogEv(EL_Wrn,EO_DOOR,1,1,'Centrale_termica_Open');
END_IF*)

(*### DOOR02 Status Check ###*)(*
fKEY_SCT_ST(IN:=KEY_SCT_ST);
IF fKEY_SCT_ST.EVH THEN
	LogEv(EL_Log,EO_DOOR,2,2,'Sottocentrale_termica_Close');
END_IF
IF fKEY_SCT_ST.EVL THEN
	LogEv(EL_Wrn,EO_DOOR,2,1,'Sottocentrale_termica_Open');
END_IF*)

(*### DOOR03 Status Check ###
fKEY_QE_ST(IN:=KEY_QE_ST);
IF fKEY_QE_ST.EVH THEN
	LogEv(EL_Log,EO_DOOR,3,2,'Quadro_Close');
END_IF
IF fKEY_QE_ST.EVL THEN
	LogEv(EL_Wrn,EO_DOOR,3,1,'Quadro_Open');
END_IF

*)
END_PROGRAM

(* POU Utils Functions/FLT_TAP, ST *)
FUNCTION_BLOCK FLT_TAP
VAR_INPUT
	IN		: BOOL;
	TAP		: BYTE:=4;
	INITEV	: BOOL:=TRUE;
END_VAR
VAR_OUTPUT
	OUT		: BOOL;
	EVH		: BOOL;
	EVL		: BOOL;
END_VAR
VAR
	init	: BOOL:=FALSE;
	cnt		: BYTE;
END_VAR
EVH:=FALSE;
EVL:=FALSE;

IF NOT init THEN
	init := TRUE;
	IF INITEV THEN
		OUT  := NOT IN;
		cnt  := TAP;
	ELSE
		OUT  := IN;
	END_IF
END_IF

IF OUT<>IN THEN
	cnt:=cnt+1;
	IF cnt>TAP THEN
		OUT:=IN;
		cnt:=0;
		IF OUT THEN EVH:=TRUE; ELSE EVL:=TRUE; END_IF
	END_IF
ELSE
	cnt:=0;
END_IF
END_FUNCTION_BLOCK

(* POU Utils Functions/ADDSTRING, ST *)
FUNCTION ADDSTRING : BOOL (* Append string to a byte buffer *)
VAR_INPUT
	pTxData: POINTER TO BYTE;
	pString: POINTER TO BYTE;
END_VAR
VAR_IN_OUT
	TxLen: DINT;
END_VAR
VAR
END_VAR
pTxData:=pTxData+TxLen;
WHILE pString^<>0 DO
	pTxData^:=pString^;
	pString:=pString+1;
	pTxData:=pTxData+1;
	TxLen:=TxLen+1;
END_WHILE
END_FUNCTION

(* POU Utils Functions/AVERAGE_T, ST *)
FUNCTION_BLOCK AVERAGE_T
VAR_INPUT
	IN: 	INT;
END_VAR
VAR_OUTPUT
	HI:		INT;
	AVG:	INT;
	LOW:	INT;
	ERR:	BOOL;
END_VAR
VAR
	sum:	DINT;
	cnt:	WORD;
END_VAR
IF cnt>=65000 THEN
	ERR:=TRUE;
	Read();
	sum := sum - AVG;
	cnt := cnt + 1;
END_IF

sum := sum + IN;
cnt := cnt + 1;

IF IN<LOW THEN  LOW:=IN; END_IF
IF IN>HI  THEN HI :=IN; END_IF
END_FUNCTION_BLOCK
ACTION Read:
AVG := DINT_TO_INT(sum/cnt);
END_ACTION
ACTION Reset:
HI:=IN;
AVG:=IN;
LOW:=IN;
ERR:=FALSE;

sum:=IN;
cnt:=1;
END_ACTION

(* POU Utils Functions/BUILD_16TO32, ST *)
FUNCTION BUILD_16TO32 : DWORD
VAR_INPUT
		pSource	:	POINTER TO WORD;
END_VAR
VAR
		Data	:	DWORD;
END_VAR
Data := WORD_TO_DWORD(pSource^);
pSource := pSource + 1;
Data := Data + WORD_TO_DWORD(pSource^) * 65536;

BUILD_16TO32 := Data;
END_FUNCTION

(* POU Utils Functions/COPY_32SWAP16, ST *)
FUNCTION COPY_32SWAP16:BOOL
VAR_INPUT
	pSourceAddress		:POINTER TO ARRAY[1..2] OF WORD;
	pDestinationAddress	:POINTER TO ARRAY[1..2] OF WORD;
END_VAR
VAR
END_VAR
pDestinationAddress^[1]:=pSourceAddress^[2];
pDestinationAddress^[2]:=pSourceAddress^[1];
END_FUNCTION

(* POU Utils Functions/FLT_EVENT, ST *)
FUNCTION_BLOCK FLT_EVENT
VAR_INPUT
	IN		: BOOL;
	INITEV	: BOOL:=TRUE;
END_VAR
VAR_OUTPUT
	EVH		: BOOL;
	EVL		: BOOL;
END_VAR
VAR
	init	: BOOL:=FALSE;
	old		: BOOL;
END_VAR
EVH:=FALSE;
EVL:=FALSE;

IF NOT init THEN
	init:=TRUE;
	IF INITEV THEN
		old := NOT IN;
	ELSE
		old := IN;
	END_IF
END_IF

IF old<>IN THEN
	old:=IN;
	IF IN THEN EVH:=TRUE; ELSE EVL:=TRUE; END_IF
END_IF
END_FUNCTION_BLOCK

(* POU Utils Functions/FLT_TIME, ST *)
FUNCTION_BLOCK FLT_TIME
VAR_INPUT
	IN		: BOOL;
	TTAP	: TIME:=T#5s;
	INITEV	: BOOL:=TRUE;
END_VAR
VAR_OUTPUT
	OUT		: BOOL;
	EVH		: BOOL;
	EVL		: BOOL;
END_VAR
VAR
	init	: BOOL:=FALSE;
	timer	: TON;
END_VAR
EVH:=FALSE;
EVL:=FALSE;

IF NOT init THEN
	init := TRUE;
	IF INITEV THEN
		OUT  := NOT IN;
	ELSE
		OUT  := IN;
	END_IF
END_IF

IF OUT<>IN THEN
	timer(IN:=TRUE,PT:=TTAP);
	IF timer.Q THEN
		OUT:=IN;
		timer(IN:=FALSE);
		IF OUT THEN EVH:=TRUE; ELSE EVL:=TRUE; END_IF
	END_IF
ELSE
	timer(IN:=FALSE);
END_IF
END_FUNCTION_BLOCK

(* POU Utils Functions/LINEAR, ST *)
FUNCTION LINEAR : REAL (* Linear interpolation *)
VAR_INPUT
	X_In	: REAL;
	P1_X	: REAL;
	P1_Y	: REAL;
	P2_X	: REAL;
	P2_Y	: REAL;
END_VAR
VAR
END_VAR
LINEAR:=P1_Y+(((P2_Y-P1_Y)*(X_In-P1_X))/(P2_X-P1_X));
END_FUNCTION

(* POU TCP_Logger/LogEv, ST *)
FUNCTION LogEv : BOOL
VAR_INPUT
	Level	: en_Logger_ErrLev;
	Object  : en_SYS_Objects;
	Index	: WORD;
	Error	: WORD;
	Message : STRING;
END_VAR
VAR
	s1 : STRING(160);
	i  : INT;
END_VAR
(* Execute error level operations *)
CASE Level OF
	EL_Wrn: 		Sys.Warning:=TRUE;
	EL_Alarm: 		Sys.Alarm  :=TRUE;
	EL_AlarmStop: 	Sys.Alarm  :=TRUE; (* GO TO STOP STATE!! *)
END_CASE

(* Fill lastlog list *)
s1:=CONCAT(Sys.Time_LogString,';Lev=');
s1:=CONCAT(s1,INT_TO_STRING(Level));
s1:=CONCAT(s1,';Obj=');
s1:=CONCAT(s1,INT_TO_STRING(Object));
s1:=CONCAT(s1,';Idx=');
s1:=CONCAT(s1,WORD_TO_STRING(Index));
s1:=CONCAT(s1,';Err=');
s1:=CONCAT(s1,WORD_TO_STRING(Error));
Sys.LastLogs_Dat[Sys.LastLogs_Idx]:=s1;
Sys.LastLogs_Msg[Sys.LastLogs_Idx]:=Message;
Sys.LastLogs_Idx:=Sys.LastLogs_Idx+1;
IF Sys.LastLogs_Idx>5 THEN Sys.LastLogs_Idx:=0; END_IF

(*---------------------------------------------------------------*)
	Logger_Head();
(*---------------------------------------------------------------*)

(* Insert ERR *)
s1:=CONCAT('&ERR=',INT_TO_STRING(Level));
s1:=CONCAT(s1,';');
s1:=CONCAT(s1,INT_TO_STRING(Object));
s1:=CONCAT(s1,';');
s1:=CONCAT(s1,WORD_TO_STRING(Index));
s1:=CONCAT(s1,';');
s1:=CONCAT(s1,WORD_TO_STRING(Error));
s1:=CONCAT(s1,';');
ADDSTRING(ADR(Logger.TData), ADR(s1), Logger.TLen);
s1:=Message;
STR_NOSPACES(ADR(s1));
ADDSTRING(ADR(Logger.TData), ADR(s1), Logger.TLen);

(*---------------------------------------------------------------*)
	Logger_Send();
(*---------------------------------------------------------------*)
END_FUNCTION

(* POU TCP_Logger/Logger_Head, ST *)
FUNCTION Logger_Head : BOOL
VAR
	s1 : STRING(160);
	i  : BYTE;
END_VAR
Logger.TLen:=0;
(* Set GET header *)
ADDSTRING(ADR(Logger.TData), ADR(Logger_GETSTART), Logger.TLen);

(* Insert Header *)
s1:=INSERT('ID=&V=1&D=',DWORD_TO_STRING(Plant_SN),3);
s1:=CONCAT(s1,Sys.Time_LogString);
s1:=CONCAT(s1,'&S=');
IF Sys.Alarm THEN i:=2; ELSIF Sys.Warning THEN i:=1; ELSE i:=0; END_IF
s1:=CONCAT(s1,BYTE_TO_STRING(i));
ADDSTRING(ADR(Logger.TData), ADR(s1), Logger.TLen);
END_FUNCTION

(* POU Utils Functions/STR_NOSPACES, ST *)
FUNCTION STR_NOSPACES : BOOL (* Replace spaces and bad chars with allowed ones, used as HTTP-GET validator *)
VAR_INPUT
	pString: POINTER TO BYTE;
END_VAR
VAR
END_VAR
WHILE pString^<>0 DO
	IF pString^=16#20 (* space *) THEN pString^:=16#5F; (*'_'*) END_IF
	pString:=pString+1;
END_WHILE
END_FUNCTION

(* POU TCP_Logger/Logger_Send, ST *)
FUNCTION Logger_Send : BOOL
VAR
	hFile: 	DWORD;
	pos:	DWORD;
END_VAR
(* Finalize string *)
ADDSTRING(ADR(Logger.TData), ADR(Logger_GETEND), Logger.TLen);

(* Read log position *)
pos:=SysFileGetSize(Logger_DataFile);
(* Check log size, bckup and erase if no pending messages *)
IF pos>5000000(*5M*) THEN
	hFile:=SysFileOpen(Logger_IndexFile,'r');
	IF hFile=0 THEN
		SysFileDelete(Logger_DataFileOld);
		SysFileRename(Logger_DataFile,Logger_DataFileOld);
		pos:=0;
	ELSE
		SysFileClose(hFile);
	END_IF
END_IF
(* Write message on log file *)
hFile:=SysFileOpen(Logger_DataFile,'a');
IF hFile<>0 THEN
	SysFileWrite(hFile, ADR(Logger.TData), Logger.TLen);
	SysFileClose(hFile);
ELSE
	Sys.Warning:=TRUE;
END_IF


(* Check logger status *)
IF Logger.SendReq=FALSE THEN
	(* Set log position for recovery *)
	Logger.SendIdx:=pos;
	(* Copy message data *)
	MEMCPY(ADR(Logger.TData),ADR(Logger.SendData),DINT_TO_WORD(Logger.TLen));
	Logger.SendLen:=Logger.TLen;
	(* Trigger request *)
	Logger.SendReq:=TRUE;
ELSE
	(* Add message position+size in recovery indexes *)
	hFile:=SysFileOpen(Logger_IndexFile,'a');
	SysFileWrite(hFile, ADR(pos), SIZEOF(pos));
	SysFileWrite(hFile, ADR(Logger.TLen), SIZEOF(Logger.TLen));
	SysFileClose(hFile);
END_IF
END_FUNCTION

(* POU Utils Functions/MEMCPY, ST *)
FUNCTION MEMCPY:BOOL
VAR_INPUT
	pSourceAddress:POINTER TO ARRAY[1..2] OF BYTE;
	pDestinationAddress:POINTER TO ARRAY[1..2] OF BYTE;
	BytesToCopy:WORD;
END_VAR
VAR
END_VAR
WHILE (BytesToCopy > 0) DO
	pDestinationAddress^[1]:=pSourceAddress^[1]; (* copy bytes from source to destination *)
	pDestinationAddress:=ADR(pDestinationAddress^[2]); (* increment destination *)
	pSourceAddress:=ADR(pSourceAddress^[2]);(* increment source *)
	BytesToCopy:=BytesToCopy -1; (* decrement number of bytes to copy *)
END_WHILE
END_FUNCTION

(* POU TCP_Logger/LogTrig, ST *)
FUNCTION LogTrig : BOOL
VAR
	s1 : STRING(160);
	i, x  : BYTE;
	w_x: WORD;
END_VAR
VAR_INPUT
END_VAR
(*---------------------------------------------------------------*)
	Logger_Head();
(*---------------------------------------------------------------*)



(* GRU01.AddLogData(CLIM:=GRU01_Clima); *)


(*
VRD01.AddLogData(CLIM:=VRD01_Clima);
VRD02.AddLogData(CLIM:=VRD02_Clima);
VRD03.AddLogData(CLIM:=VRD03_Clima); *)

FOR x:= 1 TO MAXLUM DO
	LumList[x].AddLogData;
END_FOR

(* Log LUXM *)
FOR w_x := 1 TO MAX_LUXNUM DO
	IF LuxElement[w_x].ID <> 0
	THEN LuxElement[w_x].AddLogData(LocalWorkingTime:=GlobalWorkingTime[w_x], LocalPowerOnCycles:=GlobalPowerOnCycles[w_x],
					   LocalEnergyCounter:=GlobalEnergyCounter[w_x], LocalEnergyCounter_t:=GlobalEnergyCounter_t[w_x]);
 	END_IF
END_FOR

(*
THER01.AddLogData();
THER02.AddLogData();
THER03.AddLogData();
THER04.AddLogData();
THER05.AddLogData();
*)

(*---------------------------------------------------------------*)
	Logger_Send();
(*---------------------------------------------------------------*)
END_FUNCTION

(* POU Utils Functions/MEAN_T, ST *)
FUNCTION MEAN_T : INT
VAR_INPUT
		T1		:	INT;
		T2		:	INT;

		THR_L	:	INT;
		THR_H	:	INT;
END_VAR
VAR
		Tmean	:	INT;
END_VAR
IF T1 >= THR_L AND T1 <= THR_H THEN

	IF T2 >= THR_L AND T2 <= THR_H THEN
		Tmean := (T1 + T2)/2;
	ELSE
		Tmean := T1;
	END_IF
ELSE
	IF T2 >= THR_L AND T2 <= THR_H THEN
		Tmean := T2;
	ELSE
		Tmean := 16#7FFF;	(* No valid temperature data has been passed *)
	END_IF
END_IF

MEAN_T := Tmean;
END_FUNCTION

(* POU Utils Functions/MEMCLR, ST *)
FUNCTION MEMCLR:BOOL
VAR_INPUT
	pDestinationAddress:POINTER TO ARRAY[1..2] OF BYTE;
	BytesToClear:WORD;
END_VAR
VAR
END_VAR
WHILE (BytesToClear > 0) DO
	pDestinationAddress^[1]:=0;
	pDestinationAddress:=ADR(pDestinationAddress^[2]); (* increment destination *)
	BytesToClear:=BytesToClear -1; (* decrement number of bytes to copy *)
END_WHILE
END_FUNCTION

(* POU Plant_Objects/obj_CRON, ST *)
FUNCTION_BLOCK obj_CRON
(* === CRONOGRAFO STANDARD ===
   v1.0[16/04/15] - Versioning
   v1.1[19/05/15] - Removed DB creation from previous year
*)
VAR_INPUT
	(* Settings *)
	ID			: WORD;		(* Index of instanced object *)

	InitOK		: BOOL;
	Alarm		: BOOL;
	Warning		: BOOL;

	Profile		: typ_Cron_Profile; 				(* Profilo attivo *)
	ProfileNr	: BYTE;								(* Indice profilo attivo *)
	CalendarIdx : WORD;								(* Indice calendario attivo *)
	Jolly		: ARRAY[0..9] OF typ_Cron_Jolly;	(* Jolly attivi *)

END_VAR
VAR_IN_OUT
END_VAR
VAR_OUTPUT
	SetPoint		: INT;
	(* Status *)
	Status_Log		: BYTE;
	Status_Vis 		: DWORD;
END_VAR
VAR
	Buf: 	ARRAY[0..512] OF BYTE; (* AVOID THIS!! *)
	hFile: 	DWORD;
	sFile: 	STRING;
	sFile2: STRING;

	i:		WORD;
	t1:		DWORD;
	t2:		BOOL;

END_VAR
(* Check initialization *)
IF NOT InitOK THEN Init(); END_IF

(* Chrono *)
IF CalendarIdx<>Sys.Time_CT_Day THEN DB_Load(); END_IF
SetPoint:=Profile.Setpoint[Sys.Time_CT_Minute];

(* Check jolly *)
FOR i := 0 TO 9 DO
	IF ( DT_TO_DWORD(Jolly[i].Start)>0  AND Jolly[i].End>Jolly[i].Start AND
	     Jolly[i].Start<=Sys.Time_CT_DT AND Jolly[i].End>Sys.Time_CT_DT ) THEN
			SetPoint:=Jolly[i].Temp;
	END_IF
END_FOR


(* Status color *)
   IF Alarm   THEN Status_Log:=2; Status_Vis:=COLOR_RED;
ELSIF Warning THEN Status_Log:=1; Status_Vis:=COLOR_YELLOW;
              ELSE Status_Log:=0; Status_Vis:=COLOR_GREEN;
			  END_IF
END_FUNCTION_BLOCK
ACTION AddLogData:
Logger.s1:=INSERT('&CRON=',WORD_TO_STRING(ID),5);
IF ID<10 THEN Logger.s1:=INSERT(Logger.s1,'0',5); END_IF

Logger.s1:=CONCAT(Logger.s1,INT_TO_STRING(SetPoint));			Logger.s1:=CONCAT(Logger.s1,';');

Logger.s1:=CONCAT(Logger.s1,WORD_TO_STRING(Status_Log));
ADDSTRING(ADR(Logger.TData), ADR(Logger.s1), Logger.TLen);
END_ACTION
ACTION DB_Create:
(*
(* Check presence of previous year *)
sFile2:=REPLACE(STR1:=sFile, STR2:=WORD_TO_STRING(Sys.Time_Year-1), L:=4, P:=LEN(FilesPath)+1);
hFile:=SysFileOpen(FileName:=sFile2, Mode:='r');
IF hFile<>0 THEN
	(* Check file version and close *)
	SysFileRead(File:=hFile, Buffer:=ADR(Buf), Size:=1);
	SysFileClose(File:=hFile);
END_IF
IF hFile<>0 AND Buf[0]=1 THEN
	(* Copy file *)
	SysFileCopy(FileDest:=sFile, FileSource:=sFile2);
ELSE
*)
	(* Create empty file *)
	hFile:=SysFileOpen(FileName:=sFile, Mode:='w');

	MEMCLR(pDestinationAddress:=ADR(Buf), BytesToClear:=SIZEOF(Buf));
	FOR i := 0 TO 10239 BY 512 DO
		t1:=SysFileWrite(File:=hFile, Buffer:=ADR(Buf), Size:=512);
	END_FOR
	Buf[0]:=1;
	t2:=SysFileSetPos(File:=hFile, Pos:=0);
	t1:=SysFileWrite(File:=hFile, Buffer:=ADR(Buf), Size:=1);
	SysFileClose(File:=hFile);
(*
END_IF
*)
END_ACTION
ACTION DB_Load:
DB_SetName();

(* Open data file *)
hFile:=SysFileOpen(FileName:=sFile, Mode:='r');

(* File not found *)
IF hFile=0 THEN
	Warning:=TRUE;
	LogEv(EL_Wrn,EO_CRON,ID,1,'No_data_file');
	DB_Create();
	(* Reopen file *)
	hFile:=SysFileOpen(FileName:=sFile, Mode:='r');
	IF hfile=0 THEN
		Alarm:=TRUE;
		LogEv(EL_Alarm,EO_CRON,ID,3,'Filesystem_error');
		RETURN;
	END_IF
END_IF

(* Check version *)
SysFileRead(File:=hFile, Buffer:=ADR(Buf), Size:=1);
IF Buf[0]<>1 THEN
	IF NOT Alarm THEN
		Alarm:=TRUE;
		LogEv(EL_Alarm,EO_CRON,ID,2,'Bad_data_version');
	END_IF
	SysFileClose(File:=hFile);
	RETURN;
END_IF

(* Read Jolly data *)
t2:=SysFileSetPos(File:=hFile, Pos:=512);
t1:=SysFileRead(File:=hFile, Buffer:=ADR(Jolly), Size:=SIZEOF(Jolly));
(* Read active profile index *)
CalendarIdx:=Sys.Time_CT_Day;
t2:=SysFileSetPos(File:=hFile, Pos:=(1024+4*CalendarIdx));
t1:=SysFileRead(File:=hFile, Buffer:=ADR(ProfileNr), Size:=SIZEOF(ProfileNr));
(* Read active profile *)
t2:=SysFileSetPos(File:=hFile, Pos:=(3072+512*ProfileNr));
t1:=SysFileRead(File:=hFile, Buffer:=ADR(Profile), Size:=SIZEOF(Profile));

(* Close file and validate data *)
SysFileClose(File:=hFile);
END_ACTION
ACTION DB_SetName:
(* Create current filename 'yyyyCRnn.DAT' *)
sFile:=CONCAT(FilesPath,WORD_TO_STRING(Sys.Time_Year));
sFile:=CONCAT(STR1:=sFile, STR2:='CR');
IF ID<10 THEN
sFile:=CONCAT(STR1:=sFile, STR2:='0');
END_IF
sFile:=CONCAT(STR1:=sFile, STR2:=WORD_TO_STRING(ID));
sFile:=CONCAT(STR1:=sFile, STR2:='.DAT');
END_ACTION
ACTION Init:
DB_Load();
InitOK:=TRUE;
END_ACTION

(* POU Plant_Objects/obj_CRON_EDITOR, ST *)
FUNCTION_BLOCK obj_CRON_EDITOR
(* === EDITOR CRONOGRAFO ===
   v1.0[16/04/15] - Versioning
   v1.1[19/05/15] - Create empty profile when not found
*)
VAR_INPUT

	(* Common selections *)
	CN_Sel:			BYTE:=1;
	CN_Act:			BYTE;
	CN_YSel:		WORD:=2016;
	CN_YAct:		WORD;

	(* Profile editor *)
	PR_Sel: 		BYTE:=1;
	PR_Act:			BYTE;
	PR_TT:			REAL;
	PR:				typ_Cron_Profile;
	PR_Hour:		ARRAY [0..23,0..59] OF WORD;
	PR_Minutes:		ARRAY [0..59] OF WORD;
	(* Profile signals *)
	PR_Load:		BOOL;
	PR_Save:		BOOL;
	PR_Load_Hour:	BOOL;
	PR_Save_Hour:	BOOL;

	(* Calendar editor *)
	CA_Sel:			BYTE:=1; (* Calendar month selected *)
	CA_Act:			BYTE;    (* Calendar month active *)
	CA_DayF:		BYTE:=0;
	CA_DayL:		BYTE:=31;
	CA_TPR:			BYTE;
	CA:				typ_Cron_Calendar; (* Only used for first 32 entries *)

	HourSelected		:BYTE;

	(* Calendar signals *)
	CA_Load:		BOOL;
	CA_Save:		BOOL;

	(* Jolly editor *)
	JL:				ARRAY[0..9] OF typ_Cron_Jolly;
	(* Jolly signals *)
	JL_Load:		BOOL;
	JL_Save:		BOOL;

END_VAR
VAR_OUTPUT
	Message		: STRING;
END_VAR
VAR
	sFileName	: STRING;
	sFileMode	: STRING;
	hFile		: DWORD;
	Buf			: ARRAY[0..512] OF BYTE; (* AVOID THIS!! *)

	i			: WORD;
	ver			: BYTE;
	r1			: BOOL;
	r2			: DWORD;
	x, y			:BYTE;
END_VAR
IF PR_Load THEN PR_Load_Exe(); PR_Load:=FALSE; END_IF
IF PR_Save THEN PR_Save_Exe(); PR_Save:=FALSE; END_IF
IF CA_Load THEN CA_Load_Exe(); CA_Load:=FALSE; END_IF
IF CA_Save THEN CA_Save_Exe(); CA_Save:=FALSE; END_IF
IF JL_Load THEN JL_Load_Exe(); JL_Load:=FALSE; END_IF
IF JL_Save THEN JL_Save_Exe(); JL_Save:=FALSE; END_IF
IF PR_Load_Hour THEN PR_Load_Hour_Exe(); PR_Load_Hour:=FALSE; END_IF
IF PR_Save_Hour THEN PR_Save_Hour_Exe(); PR_Save_Hour:=FALSE; END_IF
END_FUNCTION_BLOCK
ACTION CA_Load_Exe:
sFileMode:='r';
FileOpen();

IF hFile<>0 THEN

	(* Read calendar month *)
	FOR i := 0 TO 31 DO
		r1:=SysFileSetPos(File:=hFile, Pos:=(1024 + ((CA_Sel-1)*32 + i)*4));
		r2:=SysFileRead(File:=hFile, Buffer:=ADR(CA.Profile[i]), Size:=1);
	END_FOR

	(* Close file *)
	SysFileClose(File:=hFile);

	(* Validate data *)
	CA_Act :=CA_Sel;
	CN_Act :=CN_Sel;
	CN_YAct:=CN_YSel;

	Message:='Calendar load OK';

END_IF
END_ACTION
ACTION CA_Save_Exe:
sFileMode:='a';
FileOpen();

IF hFile<>0 THEN

	(* Write calendar month *)
	FOR i := 0 TO 31 DO
		r1:=SysFileSetPos(File:=hFile, Pos:=(1024 + ((CA_Sel-1)*32 + i)*4));
		r2:=SysFileGetPos(hFile);
		r2:=SysFileWrite(File:=hFile, Buffer:=ADR(CA.Profile[i]), Size:=1);
	END_FOR

	(* Close file *)
	SysFileClose(File:=hFile);

	Message:='Calendar save OK';

END_IF
END_ACTION
ACTION FileOpen:
(* Create current filename 'yyyyCRnn.DAT' *)
sFileName:=CONCAT(FilesPath,WORD_TO_STRING(CN_YSel));
sFileName:=CONCAT(STR1:=sFileName, STR2:='CR');
IF CN_Sel<10 THEN
sFileName:=CONCAT(STR1:=sFileName, STR2:='0');
END_IF
sFileName:=CONCAT(STR1:=sFileName, STR2:=BYTE_TO_STRING(CN_Sel));
sFileName:=CONCAT(STR1:=sFileName, STR2:='.DAT');

(* Check file version and size! *)
(* ... *)

(* Open data file *)
hFile:=SysFileOpen(FileName:=sFileName, Mode:='r');

(* File not found *)
IF hFile=0 THEN
	Message:='File not found - created empty file';
	(* Create empty file *)
	hFile:=SysFileOpen(FileName:=sFileName, Mode:='w');
	MEMCLR(pDestinationAddress:=ADR(Buf), BytesToClear:=SIZEOF(Buf));
	FOR i := 0 TO 10239 BY 512 DO
		SysFileWrite(File:=hFile, Buffer:=ADR(Buf), Size:=512);
	END_FOR
	Buf[0]:=1;
	SysFileSetPos(File:=hFile, Pos:=0);
	SysFileWrite(File:=hFile, Buffer:=ADR(Buf), Size:=1);
END_IF

(* Close file *)
SysFileClose(File:=hFile);

(* Open data file *)
hFile:=SysFileOpen(FileName:=sFileName, Mode:=sFileMode);
END_ACTION
ACTION JL_Load_Exe:
sFileMode:='r';
FileOpen();

IF hFile<>0 THEN

	(* Read jolly *)
	r1:=SysFileSetPos(File:=hFile, Pos:=512);
	r2:=SysFileRead(File:=hFile, Buffer:=ADR(JL), Size:=SIZEOF(JL));

	(* Close file *)
	SysFileClose(File:=hFile);

	(* Validate data *)
	CN_Act:=CN_Sel;
	CN_YAct:=CN_YSel;

	Message:='Jolly load OK';

END_IF
END_ACTION
ACTION JL_Save_Exe:
sFileMode:='a';
FileOpen();

IF hFile<>0 THEN

	(* Write selected profile *)
	r1:=SysFileSetPos(File:=hFile, Pos:=512);
	r2:=SysFileWrite(File:=hFile, Buffer:=ADR(JL), Size:=SIZEOF(JL));

	(* Close file *)
	SysFileClose(File:=hFile);

	Message:='Jolly save OK';

END_IF
END_ACTION
ACTION PR_Load_Exe:
sFileMode:='r';
FileOpen();

IF hFile<>0 THEN

	(* Read selected profile *)
	r1:=SysFileSetPos(File:=hFile, Pos:=(3072 + 512*PR_Sel));
	r2:=SysFileRead(File:=hFile, Buffer:=ADR(PR), Size:=SIZEOF(PR));

	(* Close file *)
	SysFileClose(File:=hFile);

	(* CronEd.MinSel:= CronEd.HourSelected * 60  *)

	(* Validate data *)
	PR_Act:=PR_Sel;
	CN_Act:=CN_Sel;
	CN_YAct:=CN_YSel;

	Message:='Profile load OK';

END_IF
END_ACTION
ACTION PR_Load_Hour_Exe:
sFileMode:='r';
FileOpen();

IF hFile<>0 THEN

	(* Read selected profile *)
	r1:=SysFileSetPos(File:=hFile, Pos:=(3072 + 512*PR_Sel));
	r2:=SysFileRead(File:=hFile, Buffer:=ADR(PR), Size:=SIZEOF(PR));

	(* Close file *)
	SysFileClose(File:=hFile);

	FOR x:= 0 TO 23 DO
		FOR y:= 0 TO 59 DO
			PR_Hour[x,y]:=PR.Setpoint[y+(60*x)];
		END_FOR
	END_FOR
	FOR x:= 0 TO 59 DO
		PR_Minutes[x]:=PR_Hour[HourSelected,x];
	END_FOR
	(* CronEd.MinSel:= CronEd.HourSelected * 60  *)

	(* Validate data *)
	PR_Act:=PR_Sel;
	CN_Act:=CN_Sel;
	CN_YAct:=CN_YSel;

	Message:='Profile load OK';

END_IF
END_ACTION
ACTION PR_Save_Exe:
sFileMode:='a';
FileOpen();

IF hFile<>0 THEN

	(* Write selected profile *)
	r1:=SysFileSetPos(File:=hFile, Pos:=(3072 + 512*PR_Sel));
	r2:=SysFileWrite(File:=hFile, Buffer:=ADR(PR), Size:=SIZEOF(PR));

	(* Close file *)
	SysFileClose(File:=hFile);

	Message:='Profile save OK';

END_IF
END_ACTION
ACTION PR_Save_Hour_Exe:
sFileMode:='a';
FileOpen();

IF hFile<>0 THEN

	FOR x:= 0 TO 59 DO
		PR_Hour[HourSelected,x]:=PR_Minutes[x];
	END_FOR
	FOR y:= 0 TO 59 DO
		PR.Setpoint[y+(60*HourSelected)]:=PR_Hour[HourSelected,y];
	END_FOR
	(* Write selected profile *)
	r1:=SysFileSetPos(File:=hFile, Pos:=(3072 + 512*PR_Sel));
	r2:=SysFileWrite(File:=hFile, Buffer:=ADR(PR), Size:=SIZEOF(PR));

	(* Close file *)
	SysFileClose(File:=hFile);

	Message:='Profile save OK';

END_IF
END_ACTION

(* POU Plant_Objects/obj_CRONTER, ST *)
FUNCTION_BLOCK obj_CRONTER
(* === THERMOSTAT ===
   v1.0[30/07/15] - Versioning
*)
VAR_INPUT
	(* Settings *)
	ID			: BYTE;		(* Index of instanced object *)

	InitOK		: BOOL;
	Alarm		: BOOL;
	Warning		: BOOL;

	Profile		: typ_Cron_Profile; 				(* Profilo attivo *)
	ProfileNr	: BYTE;								(* Indice profilo attivo *)
	CalendarIdx : WORD;								(* Indice calendario attivo *)
	Jolly		: ARRAY[0..9] OF typ_Cron_Jolly;	(* Jolly attivi *)

	Temperature	: INT;
	Local_MaxRunTAmb	:	INT;					(* Local maximum environment temperature, NOT "TAMB" *)
	Histeresys:INT; (* isteresi per la ripartenza del Comando ON*)


END_VAR
VAR_IN_OUT
END_VAR
VAR_OUTPUT
	SetPoint		: INT;
	Run				: BOOL;
	AntifreezeForce	: BOOL;
	RunCrono		: BOOL;

	(* Status *)
	Status_Log		: BYTE;
	Status_Vis 		: DWORD;
END_VAR
VAR
	Buf: 	ARRAY[0..512] OF BYTE; (* AVOID THIS!! *)
	hFile: 	DWORD;
	sFile: 	STRING;
	sFile2: STRING;

	i:		WORD;
	t1:		DWORD;
	t2:		BOOL;

END_VAR
(* Check initialization *)
IF NOT InitOK THEN Init(); END_IF

(* Check Temperature *)
IF Temperature <Local_MaxRunTAmb THEN

	(* LOCAL environment temperature lower than maximum allowed -> Proceed with SetPoint adjustment *)
	(* Chrono *)
	IF CalendarIdx<>Sys.Time_CT_Day THEN DB_Load(); END_IF
	SetPoint:=Profile.Setpoint[Sys.Time_CT_Quarter];

	(* Check jolly *)
	FOR i := 0 TO 9 DO
		IF ( DT_TO_DWORD(Jolly[i].Start)>0  AND Jolly[i].End>Jolly[i].Start AND
		     Jolly[i].Start<=Sys.Time_CT_DT AND Jolly[i].End>Sys.Time_CT_DT ) THEN
				SetPoint:=Jolly[i].Temp;
		END_IF
	END_FOR

(*
	IF SetPoint < 180 THEN
		(* Switch off the device *)
		Run := FALSE;
	ELSE
		(* Set according to feedback T - Histeresys of 1°C *)
		IF Temperature >= (SetPoint + 5) THEN
			Run := FALSE;
		ELSIF Temperature <= (SetPoint - 5) THEN
			Run := TRUE;
		END_IF

		(* Between "SetPoint-5" and "SetPoint+5" last state (ON or OFF) of "Run" is kept	*)
	END_IF
*)
(* Gestione uscita Crono *)
		IF SetPoint>0 THEN RunCrono := TRUE;
		ELSIF SetPoint=0 THEN RunCrono := FALSE;
		END_IF

(* GEstione uscita Cronotermostato *)

		IF Temperature >= (SetPoint) THEN
			Run := FALSE;
		ELSIF Temperature <= (SetPoint - Histeresys) THEN
			Run := TRUE;
		END_IF
ELSE
	(* Environment overtemperature: stop heating -> Stop device *)
	Run := FALSE;
END_IF

(* Freeze warning: Switch on and heat! *)
(*IF Temperature < Plant_AntiFreezeTAmb THEN AntifreezeForce := TRUE;
ELSE AntifreezeForce := FALSE;
END_IF*)



(* Status color *)
   IF Alarm   THEN Status_Log:=2; Status_Vis:=COLOR_RED;
ELSIF Warning THEN Status_Log:=1; Status_Vis:=COLOR_YELLOW;
              ELSE Status_Log:=0; Status_Vis:=COLOR_GREEN;
			  END_IF
END_FUNCTION_BLOCK
ACTION AddLogData:
Logger.s1:=INSERT('&THER=',BYTE_TO_STRING(ID),5);
IF ID<10 THEN Logger.s1:=INSERT(Logger.s1,'0',5); END_IF

Logger.s1:=CONCAT(Logger.s1,INT_TO_STRING(SetPoint));			Logger.s1:=CONCAT(Logger.s1,';');

Logger.s1:=CONCAT(Logger.s1,WORD_TO_STRING(Status_Log));
ADDSTRING(ADR(Logger.TData), ADR(Logger.s1), Logger.TLen);
END_ACTION
ACTION DB_Create:
(* Create empty file *)
hFile:=SysFileOpen(FileName:=sFile, Mode:='w');

MEMCLR(pDestinationAddress:=ADR(Buf), BytesToClear:=SIZEOF(Buf));
FOR i := 0 TO 10239 BY 512 DO
	t1:=SysFileWrite(File:=hFile, Buffer:=ADR(Buf), Size:=512);		(* Clear created file (all bytes 0) *)
END_FOR
Buf[0]:=1;
t2:=SysFileSetPos(File:=hFile, Pos:=0);
t1:=SysFileWrite(File:=hFile, Buffer:=ADR(Buf), Size:=1);
SysFileClose(File:=hFile);
END_ACTION
ACTION DB_Load:
DB_SetName();

(* Open data file *)
hFile:=SysFileOpen(FileName:=sFile, Mode:='r');

(* File not found *)
IF hFile=0 THEN
	Warning:=TRUE;
	LogEv(EL_Wrn,EO_CRON,ID,1,'No_data_file');
	DB_Create();
	(* Reopen file *)
	hFile:=SysFileOpen(FileName:=sFile, Mode:='r');
	IF hfile=0 THEN
		Alarm:=TRUE;
		LogEv(EL_Alarm,EO_CRON,ID,3,'Filesystem_error');
		RETURN;
	END_IF
END_IF

(* Check version *)
SysFileRead(File:=hFile, Buffer:=ADR(Buf), Size:=1);
IF Buf[0]<>1 THEN
	IF NOT Alarm THEN
		Alarm:=TRUE;
		LogEv(EL_Alarm,EO_CRON,ID,2,'Bad_data_version');
	END_IF
	SysFileClose(File:=hFile);
	RETURN;
END_IF

(* Read Jolly data *)
t2:=SysFileSetPos(File:=hFile, Pos:=512);
t1:=SysFileRead(File:=hFile, Buffer:=ADR(Jolly), Size:=SIZEOF(Jolly));
(* Read active profile index *)
CalendarIdx:=Sys.Time_CT_Day;
t2:=SysFileSetPos(File:=hFile, Pos:=(1024+4*CalendarIdx));
t1:=SysFileRead(File:=hFile, Buffer:=ADR(ProfileNr), Size:=SIZEOF(ProfileNr));
(* Read active profile *)
t2:=SysFileSetPos(File:=hFile, Pos:=(3072+512*ProfileNr));
t1:=SysFileRead(File:=hFile, Buffer:=ADR(Profile), Size:=SIZEOF(Profile));

(* Close file and validate data *)
SysFileClose(File:=hFile);
END_ACTION
ACTION DB_SetName:
(* Create current filename 'yyyyCRnn.DAT' *)
sFile:=CONCAT(FilesPath,WORD_TO_STRING(Sys.Time_Year));
sFile:=CONCAT(STR1:=sFile, STR2:='CR');
IF ID<10 THEN
sFile:=CONCAT(STR1:=sFile, STR2:='0');
END_IF
sFile:=CONCAT(STR1:=sFile, STR2:=BYTE_TO_STRING(ID));
sFile:=CONCAT(STR1:=sFile, STR2:='.DAT');
END_ACTION
ACTION Init:
DB_Load();
InitOK:=TRUE;
END_ACTION

(* POU Plant_Objects/obj_LUM, ST *)
FUNCTION_BLOCK obj_LUM (*  Lux probe *)
VAR CONSTANT
	NormalEv		: BYTE := 0;
	ErrorEv			: BYTE := 1;
	WarningEv		: BYTE := 2;

END_VAR

VAR_INPUT
	ID				: BYTE;
	TAP				: BYTE:=4;	   (* Consecutive checks filter *)


	INITEV			: BOOL:= TRUE; (* Generate init OK event *)
	IN_EMIN_lux		: INT:=1;	(*  INT *)(*   Low error limit in lux  *) (* 50  *)
	IN_EMIN			: DWORD; 	(*   Low error limit in bit  *) (* era Int *)

	IN_WMIN_lux	: INT := 100; 	(*  INT *) (* Low warning value in lux  *) (* 100  *)
	IN_WMIN		: DWORD;		 (* Low warning value in bit  *) (* era Int *)
	IN_WMAX_lux	: DWORD :=  850; 	(*  DWORD *)  (* High warning value in lux  *) (* 80000  *)
	IN_WMAX		: DWORD;		 (* Low warning value in bit  *)  (* era Int *)
	IN_EMAX_lux		: DWORD := 900; 	(*  DWORD *)  (* High error limit in lux *) (* 99000  *)
	IN_EMAX			: DWORD;  (* High error limit in bit *)  (* era Int *)

	ERR_MIN_SHORT	: BOOL:= TRUE; (* TRUE  ==> EMIN=Short        , EMAX=Disconnected
									  FALSE ==> EMIN=Disconnected , EMAX=Short 		 *)
	IN_TARGET		: INT;

	(* Physical input *)
	IN			: INT;
END_VAR

VAR_OUTPUT
	WRN			: BOOL;	(* Value in warning range *)
	ERR			: BOOL;	(* Value error *)
	HI			: INT;	(* Highest value - cleared by Stat_Reset() action *)
	AVG			: INT; 	(* Average value - updated by Mean() action, cleared by Mean_Reset() action *)
	LOW			: INT;	(* Lowest value  - cleared by Stat_Reset() action *)

	Status_Log	: WORD;
	Status_Vis	: DWORD;
END_VAR
VAR
	cnt			: BYTE;
	event		: BYTE := 0;	(* 0: monitoring a generic, 1: monitoring an error, 2: monitoring a warning *)
	asum		: DINT;
	acnt		: WORD;
	AVG_Lux		:INT;
END_VAR
(* Check probe value limits *)
	IN_EMIN_lux:= INT_TO_WORD((IN_TARGET-300));
	IF IN_EMIN_lux < 0 THEN IN_EMIN_lux := 0; END_IF
	IN_EMAX_lux:= INT_TO_WORD((IN_TARGET+300));
	IF IN_EMAX_lux > 1000 THEN IN_EMAX_lux := 1000; END_IF
	IN_WMIN_lux:= INT_TO_WORD((IN_TARGET- 100));
	IF IN_WMIN_lux < 0 THEN IN_WMIN_lux := 0; END_IF
	IN_WMAX_lux:= INT_TO_WORD((IN_TARGET+100));
	IF IN_WMAX_lux > 1000 THEN IN_WMAX_lux := 1000; END_IF
 
(*
	IN_EMIN_lux:= ((IN_TARGET*0.7));
	IF IN_EMIN_lux < 0 THEN IN_EMIN_lux := 0; END_IF
	IN_EMAX_lux:= ((IN_TARGET*1.3));
	IF IN_EMAX_lux > 1000 THEN IN_EMAX_lux := 1000; END_IF
	IN_WMIN_lux:= ((IN_TARGET*0.9));
	IF IN_WMIN_lux < 0 THEN IN_WMIN_lux := 0; END_IF
	IN_WMAX_lux:= ((IN_TARGET*1.1));
 *)
	IF IN_WMAX_lux > 1000 THEN IN_WMAX_lux := 1000; END_IF
IN_EMIN := REAL_TO_DWORD(IN_EMIN_lux*32.767);
IN_EMAX :=REAL_TO_DWORD (IN_EMAX_lux*32.767);
IN_WMIN := REAL_TO_DWORD(IN_WMIN_lux*32.767);
IN_WMAX := REAL_TO_DWORD(IN_WMAX_lux*32.767);


IF IN<=IN_EMIN OR IN>=IN_EMAX THEN
	IF NOT ERR THEN
		IF event <> ErrorEv THEN
			cnt := 1;
			event := ErrorEv;
		ELSE
			cnt:=cnt+1;
		END_IF

		IF cnt>TAP THEN
			cnt:=0;
			ERR:=TRUE; WRN:=FALSE;
			IF ( ERR_MIN_SHORT=TRUE  AND IN<=IN_EMIN ) OR ( ERR_MIN_SHORT=FALSE AND IN>=IN_EMAX ) THEN
				LogEv(EL_Alarm,EO_LUM,ID,5,INT_TO_STRING(IN));
			ELSE
				LogEv(EL_Alarm,EO_LUM,ID,4,INT_TO_STRING(IN));
			END_IF
		END_IF
	END_IF
ELSIF IN<=IN_WMIN OR IN>=IN_WMAX THEN
	IF NOT WRN THEN
		IF event <> WarningEv THEN
			cnt := 1;
			event := WarningEv;
		ELSE
			cnt:=cnt+1;
		END_IF

		IF cnt>TAP THEN
			cnt:=0;
			ERR:=FALSE; WRN:=TRUE;
			LogEv(EL_Wrn,EO_LUM,ID,SEL(IN<=IN_WMIN,3,2),INT_TO_STRING(IN));
		END_IF
	END_IF
ELSE
	IF INITEV OR WRN OR ERR THEN
		IF event <> NormalEv THEN
			cnt := 1;
			event := NormalEv;
		ELSE
			cnt:=cnt+1;
		END_IF

		IF cnt>TAP THEN
			cnt:=0;
			INITEV:=FALSE; ERR:=FALSE; WRN:=FALSE;
			LogEv(EL_Log,EO_LUM,ID,1,'Probe_OK');
		END_IF
	END_IF
END_IF



(* Average value *)


AVG := IN;
AVG_Lux:=REAL_TO_INT( AVG * LuxSuBit);


(* Statistics values *)
IF IN<LOW THEN LOW:=IN; END_IF
IF IN>HI  THEN HI :=IN; END_IF


(* Status Log *)
IF ERR THEN	Status_Log := 2; Status_Vis := COLOR_RED;
ELSIF WRN THEN Status_Log := 1;	Status_Vis := COLOR_YELLOW;
ELSE Status_Log := 0; Status_Vis := COLOR_GREEN;
END_IF
END_FUNCTION_BLOCK
ACTION AddLogData:
Logger.s1:=INSERT('&LUM=',BYTE_TO_STRING(ID),4);
IF ID<10 THEN Logger.s1:=INSERT(Logger.s1,'0',4); END_IF;

Logger.s1:=CONCAT(Logger.s1,INT_TO_STRING(AVG_Lux));		Logger.s1:=CONCAT(Logger.s1,';');

Logger.s1:=CONCAT(Logger.s1,WORD_TO_STRING(Status_Log));
ADDSTRING(ADR(Logger.TData), ADR(Logger.s1), Logger.TLen);
END_ACTION

(* POU Plant_Objects/obj_LUX, ST *)
FUNCTION_BLOCK obj_LUX
(*
   v1.0[feb-2016] - Create GIURE      
	
   Info:
   	
*)
VAR CONSTANT
	(*Costant in lux obj*)
	NO_DIMMING	: BYTE:=0;
	DIMMING		: BYTE:=1;
	ROT			: BOOL:=1;
	GRUN		: BOOL:=0;
END_VAR

